KUKA KRL program: MyProgram_151().src

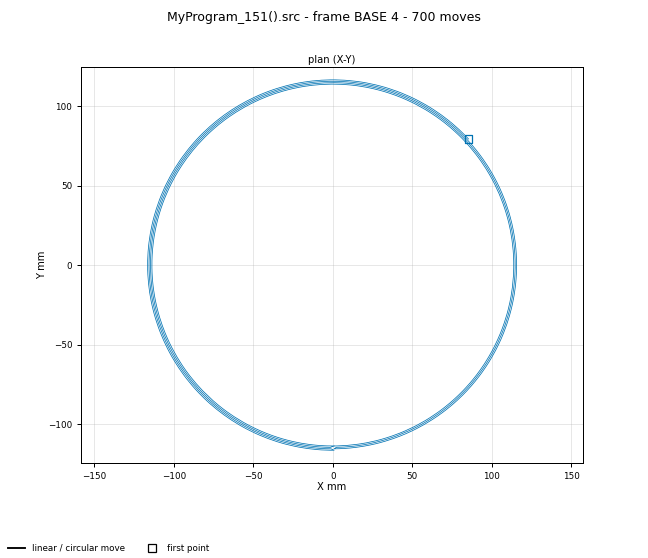
[picture p0: tool path of MyProgram_151().src in frame BASE 4, 700 of 700 moves have a stored position in this frame; points joined in program order, loops and branches not executed]
&ACCESS RVP
&REL 1
&PARAM TEMPLATE = C:\KRC\Roboter\Template\vorgabe
&PARAM EDITMASK = *
DEF MyProgram_151()
; ---- Setting reference (Base) ----
$BASE = BASE_DATA[4]

; --------------------------
; ---- Setting tool (TCP) ----
$TOOL = TOOL_DATA[3]
; --------------------------

$VEL.CP = VEL_APROX_PRINT
Startdeposition()
$VEL.CP = VEL_PRINT
LIN {X 85.3348,Y 79.272,Z 118,A 39.0033,B 24.9377,C -1.8229,E1 25.1164,E2 406.8947} C_DIS
LIN {X 83.3637,Y 81.3423,Z 118,A 40.3329,B 24.9377,C -1.8225,E1 25.1138,E2 405.572} C_DIS
LIN {X 81.214,Y 83.4873,Z 118,A 41.7921,B 24.9377,C -1.8241,E1 25.1109,E2 404.1151} C_DIS
LIN {X 79.272,Y 85.3348,Z 118,A 43.1327,B 24.9374,C -1.8278,E1 25.1082,E2 402.7712} C_DIS
LIN {X 76.7632,Y 87.5957,Z 118,A 44.7729,B 24.9372,C -1.8302,E1 25.1048,E2 401.1319} C_DIS
LIN {X 74.8522,Y 89.2356,Z 118,A 46.0205,B 24.937,C -1.833,E1 25.1021,E2 399.8825} C_DIS
LIN {X 72.6397,Y 91.0457,Z 118,A 47.421,B 24.9369,C -1.8354,E1 25.0991,E2 398.4816} C_DIS
LIN {X 70.3835,Y 92.8009,Z 118,A 48.9052,B 24.9364,C -1.8416,E1 25.0957,E2 396.9883} C_DIS
LIN {X 68.2299,Y 94.3968,Z 118,A 50.1353,B 24.9366,C -1.8398,E1 25.093,E2 395.7667} C_DIS
LIN {X 65.5697,Y 96.2615,Z 118,A 51.6474,B 24.9366,C -1.8386,E1 25.0895,E2 394.2626} C_DIS
LIN {X 63.3659,Y 97.7272,Z 118,A 53.0869,B 24.9361,C -1.847,E1 25.0861,E2 392.808} C_DIS
LIN {X 61.1008,Y 99.1603,Z 118,A 54.4098,B 24.9359,C -1.8492,E1 25.083,E2 391.4841} C_DIS
LIN {X 58.4944,Y 100.7187,Z 118,A 55.8287,B 24.9359,C -1.848,E1 25.0796,E2 390.0724} C_DIS
LIN {X 56.005,Y 102.1239,Z 118,A 57.3305,B 24.9355,C -1.8543,E1 25.0759,E2 388.56} C_DIS
LIN {X 53.6405,Y 103.3865,Z 118,A 58.5455,B 24.9358,C -1.8513,E1 25.0729,E2 387.3555} C_DIS
LIN {X 51.0872,Y 104.6717,Z 118,A 59.9607,B 24.9356,C -1.8535,E1 25.0694,E2 385.9389} C_DIS
LIN {X 48.503,Y 105.894,Z 118,A 61.3507,B 24.9356,C -1.8545,E1 25.0659,E2 384.5502} C_DIS
LIN {X 45.6034,Y 107.173,Z 118,A 62.7679,B 24.9359,C -1.8498,E1 25.0623,E2 383.1475} C_DIS
LIN {X 43.2486,Y 108.1463,Z 118,A 64.227,B 24.9351,C -1.8604,E1 25.0584,E2 381.6667} C_DIS
LIN {X 40.5815,Y 109.1751,Z 118,A 65.5599,B 24.9353,C -1.8584,E1 25.055,E2 380.3412} C_DIS
LIN {X 37.7211,Y 110.1951,Z 118,A 67.0508,B 24.9352,C -1.8596,E1 25.0511,E2 378.8505} C_DIS
LIN {X 35.1757,Y 111.0349,Z 118,A 68.4376,B 24.9349,C -1.8638,E1 25.0473,E2 377.4565} C_DIS
LIN {X 32.4402,Y 111.8647,Z 118,A 69.7714,B 24.935,C -1.8615,E1 25.0438,E2 376.1303} C_DIS
LIN {X 29.6851,Y 112.6271,Z 118,A 71.1757,B 24.935,C -1.8624,E1 25.04,E2 374.7262} C_DIS
LIN {X 26.9121,Y 113.3217,Z 118,A 72.58,B 24.935,C -1.8631,E1 25.0362,E2 373.3222} C_DIS
LIN {X 23.9484,Y 113.9839,Z 118,A 73.9931,B 24.9351,C -1.8603,E1 25.0324,E2 371.9178} C_DIS
LIN {X 21.3193,Y 114.5057,Z 118,A 75.4604,B 24.9346,C -1.8674,E1 25.0283,E2 370.4352} C_DIS
LIN {X 18.5028,Y 114.9944,Z 118,A 76.795,B 24.9348,C -1.8647,E1 25.0246,E2 369.1083} C_DIS
LIN {X 15.6751,Y 115.4139,Z 118,A 78.2709,B 24.9346,C -1.8682,E1 25.0205,E2 367.6255} C_DIS
LIN {X 12.6607,Y 115.7824,Z 118,A 79.6939,B 24.9348,C -1.8653,E1 25.0166,E2 366.2103} C_DIS
LIN {X 9.9931,Y 116.044,Z 118,A 81.1695,B 24.9343,C -1.8724,E1 25.0125,E2 364.7188} C_DIS
LIN {X 7.1422,Y 116.2543,Z 118,A 82.4182,B 24.9348,C -1.8654,E1 25.009,E2 363.4871} C_DIS
LIN {X 4.1089,Y 116.4,Z 118,A 83.9124,B 24.9348,C -1.8654,E1 25.0049,E2 361.9935} C_DIS
LIN {X 1.4293,Y 116.4647,Z 118,A 85.302,B 24.9346,C -1.8683,E1 25.001,E2 360.5972} C_DIS
LIN {X -1.4293,Y 116.4647,Z 118,A 86.6382,B 24.9348,C -1.8649,E1 24.9973,E2 359.2689} C_DIS
LIN {X -4.4651,Y 116.3869,Z 118,A 88.1333,B 24.9348,C -1.8645,E1 24.9931,E2 357.7745} C_DIS
LIN {X -7.1422,Y 116.2543,Z 118,A 89.5233,B 24.9346,C -1.8672,E1 24.9892,E2 356.378} C_DIS
LIN {X -10.1706,Y 116.0276,Z 118,A 90.9807,B 24.9348,C -1.8649,E1 24.9852,E2 354.9252} C_DIS
LIN {X -12.838,Y 115.7638,Z 118,A 92.3389,B 24.9348,C -1.8659,E1 24.9814,E2 353.5638} C_DIS
LIN {X -15.6751,Y 115.4139,Z 118,A 93.6765,B 24.935,C -1.862,E1 24.9777,E2 352.2345} C_DIS
LIN {X -18.5028,Y 114.9944,Z 118,A 95.0845,B 24.935,C -1.8611,E1 24.9738,E2 350.8273} C_DIS
LIN {X -21.3193,Y 114.5057,Z 118,A 96.4933,B 24.9351,C -1.8602,E1 24.9699,E2 349.4193} C_DIS
LIN {X -24.2971,Y 113.9101,Z 118,A 97.9106,B 24.9355,C -1.8556,E1 24.9661,E2 348.0112} C_DIS
LIN {X -27.0853,Y 113.2795,Z 118,A 99.3197,B 24.9355,C -1.8544,E1 24.9623,E2 346.6031} C_DIS
LIN {X -29.8571,Y 112.5806,Z 118,A 100.7287,B 24.9356,C -1.8532,E1 24.9585,E2 345.195} C_DIS
LIN {X -32.6721,Y 111.7959,Z 118,A 102.2246,B 24.9356,C -1.8541,E1 24.9544,E2 343.6945} C_DIS
LIN {X -35.3452,Y 110.98,Z 118,A 103.6275,B 24.9356,C -1.8537,E1 24.9507,E2 342.2901} C_DIS
LIN {X -38.0582,Y 110.0792,Z 118,A 105.0374,B 24.9356,C -1.8522,E1 24.947,E2 340.8812} C_DIS
LIN {X -40.7482,Y 109.112,Z 118,A 106.4477,B 24.9358,C -1.8505,E1 24.9433,E2 339.472} C_DIS
LIN {X -43.4137,Y 108.0791,Z 118,A 107.858,B 24.9359,C -1.8487,E1 24.9396,E2 338.0628} C_DIS
LIN {X -46.053,Y 106.9812,Z 118,A 109.2688,B 24.9361,C -1.8469,E1 24.936,E2 336.6532} C_DIS
LIN {X -48.6646,Y 105.8188,Z 118,A 110.6668,B 24.9362,C -1.8444,E1 24.9324,E2 335.2577} C_DIS
LIN {X -51.56,Y 104.4374,Z 118,A 112.0273,B 24.937,C -1.8327,E1 24.9291,E2 333.9215} C_DIS
LIN {X -53.8634,Y 103.2691,Z 118,A 113.5098,B 24.9366,C -1.8395,E1 24.9253,E2 332.4188} C_DIS
LIN {X -56.3172,Y 101.952,Z 118,A 114.9134,B 24.9366,C -1.8386,E1 24.9219,E2 331.0134} C_DIS
LIN {X -58.8023,Y 100.5392,Z 118,A 116.2454,B 24.937,C -1.8329,E1 24.9187,E2 329.6909} C_DIS
LIN {X -61.3804,Y 98.9856,Z 118,A 117.6643,B 24.9374,C -1.8276,E1 24.9153,E2 328.2803} C_DIS
LIN {X -63.5159,Y 97.631,Z 118,A 119.1322,B 24.9369,C -1.8346,E1 24.9118,E2 326.7911} C_DIS
LIN {X -66.0391,Y 95.9411,Z 118,A 120.5614,B 24.9373,C -1.8289,E1 24.9085,E2 325.3705} C_DIS
LIN {X -68.2299,Y 94.3968,Z 118,A 121.9567,B 24.9373,C -1.8294,E1 24.9054,E2 323.9693} C_DIS
LIN {X -70.6671,Y 92.5851,Z 118,A 123.3066,B 24.9379,C -1.8202,E1 24.9024,E2 322.6363} C_DIS
LIN {X -72.7796,Y 90.9352,Z 118,A 124.7114,B 24.9379,C -1.821,E1 24.8993,E2 321.2246} C_DIS
LIN {X -75.125,Y 89.0061,Z 118,A 126.2124,B 24.9381,C -1.8179,E1 24.8961,E2 319.7251} C_DIS
LIN {X -77.1539,Y 87.2545,Z 118,A 127.5376,B 24.9382,C -1.8152,E1 24.8933,E2 318.4011} C_DIS
LIN {X -79.5348,Y 85.0876,Z 118,A 128.9678,B 24.9389,C -1.8051,E1 24.8904,E2 316.9892} C_DIS
LIN {X -81.3423,Y 83.3637,Z 118,A 130.3644,B 24.9387,C -1.8091,E1 24.8875,E2 315.5773} C_DIS
LIN {X -83.3637,Y 81.3423,Z 118,A 131.8491,B 24.9387,C -1.8089,E1 24.8846,E2 314.0867} C_DIS
LIN {X -85.4553,Y 79.1407,Z 118,A 133.28,B 24.9391,C -1.8026,E1 24.8819,E2 312.6646} C_DIS
LIN {X -87.3718,Y 77.0196,Z 118,A 134.6941,B 24.9393,C -1.7993,E1 24.8793,E2 311.252} C_DIS
LIN {X -89.2356,Y 74.8522,Z 118,A 136.0285,B 24.9398,C -1.7927,E1 24.8769,E2 309.9273} C_DIS
LIN {X -90.9352,Y 72.7796,Z 118,A 137.4345,B 24.9398,C -1.7927,E1 24.8744,E2 308.5145} C_DIS
LIN {X -92.8009,Y 70.3835,Z 118,A 138.9372,B 24.94,C -1.7891,E1 24.8719,E2 307.0133} C_DIS
LIN {X -94.3968,Y 68.2299,Z 118,A 140.3345,B 24.94,C -1.7887,E1 24.8695,E2 305.6102} C_DIS
LIN {X -96.0428,Y 65.8928,Z 118,A 141.6783,B 24.9405,C -1.7822,E1 24.8674,E2 304.2753} C_DIS
LIN {X -97.7235,Y 63.3718,Z 118,A 143.1007,B 24.9409,C -1.7752,E1 24.8652,E2 302.8623} C_DIS
LIN {X -99.1603,Y 61.1008,Z 118,A 144.5079,B 24.9409,C -1.7749,E1 24.8632,E2 301.4487} C_DIS
LIN {X -100.7187,Y 58.4943,Z 118,A 146.0113,B 24.9412,C -1.771,E1 24.861,E2 299.9469} C_DIS
LIN {X -102.1239,Y 56.005,Z 118,A 147.4264,B 24.9415,C -1.7673,E1 24.8591,E2 298.5333} C_DIS
LIN {X -103.5905,Y 53.2413,Z 118,A 148.8412,B 24.9421,C -1.7576,E1 24.8573,E2 297.134} C_DIS
LIN {X -104.7489,Y 50.9265,Z 118,A 150.1771,B 24.9421,C -1.7563,E1 24.8556,E2 295.7939} C_DIS
LIN {X -105.894,Y 48.503,Z 118,A 151.5844,B 24.9422,C -1.7559,E1 24.854,E2 294.3799} C_DIS
LIN {X -107.1216,Y 45.7254,Z 118,A 153.0082,B 24.9427,C -1.7485,E1 24.8524,E2 292.966} C_DIS
LIN {X -108.1463,Y 43.2486,Z 118,A 154.4865,B 24.9425,C -1.751,E1 24.8508,E2 291.4735} C_DIS
LIN {X -109.1751,Y 40.5815,Z 118,A 155.8314,B 24.943,C -1.7441,E1 24.8495,E2 290.1375} C_DIS
LIN {X -110.1951,Y 37.7211,Z 118,A 157.335,B 24.9433,C -1.7398,E1 24.8481,E2 288.6355} C_DIS
LIN {X -111.0349,Y 35.1757,Z 118,A 158.7337,B 24.9433,C -1.7389,E1 24.8469,E2 287.2309} C_DIS
LIN {X -112.2544,Y 31.065,Z 118,A 160.8577,B 24.9437,C -1.7328,E1 24.8453,E2 285.1092} C_DIS
LIN {X -112.9829,Y 28.3007,Z 118,A 162.2735,B 24.944,C -1.7287,E1 24.8443,E2 283.695} C_DIS
LIN {X -113.6814,Y 25.3454,Z 118,A 163.7071,B 24.9445,C -1.7214,E1 24.8434,E2 282.2702} C_DIS
LIN {X -114.341,Y 22.175,Z 118,A 165.0605,B 24.9454,C -1.7065,E1 24.8427,E2 280.9443} C_DIS
LIN {X -114.7881,Y 19.7367,Z 118,A 166.4593,B 24.9452,C -1.7099,E1 24.842,E2 279.5293} C_DIS
LIN {X -115.2655,Y 16.7194,Z 118,A 168.0902,B 24.9452,C -1.7103,E1 24.8413,E2 277.8878} C_DIS
LIN {X -115.6183,Y 14.0806,Z 118,A 169.3713,B 24.9455,C -1.7048,E1 24.8408,E2 276.612} C_DIS
LIN {X -115.929,Y 11.2389,Z 118,A 170.7075,B 24.946,C -1.6974,E1 24.8405,E2 275.2856} C_DIS
LIN {X -116.1699,Y 8.3905,Z 118,A 172.1239,B 24.9463,C -1.6932,E1 24.8401,E2 273.8705} C_DIS
LIN {X -116.3408,Y 5.537,Z 118,A 173.6198,B 24.9463,C -1.6923,E1 24.8399,E2 272.3678} C_DIS
LIN {X -116.4384,Y 2.8584,Z 118,A 175.0528,B 24.9463,C -1.6927,E1 24.8399,E2 270.9254} C_DIS
LIN {X -116.4727,Y 0,Z 118,A 176.3346,B 24.9469,C -1.683,E1 24.8398,E2 269.6588} C_DIS
LIN {X -116.4384,Y -2.8584,Z 118,A 177.8509,B 24.9469,C -1.683,E1 24.8398,E2 268.1336} C_DIS
LIN {X -116.3233,Y -5.893,Z 118,A 179.2044,B 24.9476,C -1.6724,E1 24.84,E2 266.7971} C_DIS
LIN {X -116.1437,Y -8.746,Z 118,A -179.3796,B 24.9478,C -1.6682,E1 24.8403,E2 265.3825} C_DIS
LIN {X -115.9126,Y -11.4164,Z 118,A -177.9721,B 24.9478,C -1.6676,E1 24.8407,E2 263.968} C_DIS
LIN {X -115.5747,Y -14.4343,Z 118,A -176.5474,B 24.9484,C -1.66,E1 24.8411,E2 262.5529} C_DIS
LIN {X -115.2128,Y -17.0902,Z 118,A -175.14,B 24.9484,C -1.6594,E1 24.8417,E2 261.1385} C_DIS
LIN {X -114.7272,Y -20.0879,Z 118,A -173.6359,B 24.9487,C -1.6551,E1 24.8424,E2 259.6357} C_DIS
LIN {X -114.2355,Y -22.7228,Z 118,A -172.2374,B 24.9487,C -1.6543,E1 24.8431,E2 258.231} C_DIS
LIN {X -113.6434,Y -25.5195,Z 118,A -170.8217,B 24.949,C -1.6502,E1 24.844,E2 256.8166} C_DIS
LIN {X -112.9829,Y -28.3007,Z 118,A -169.406,B 24.9492,C -1.6463,E1 24.8449,E2 255.402} C_DIS
LIN {X -112.2544,Y -31.065,Z 118,A -168.0613,B 24.9496,C -1.6394,E1 24.8459,E2 254.066} C_DIS
LIN {X -111.4054,Y -33.9807,Z 118,A -166.5575,B 24.9499,C -1.6353,E1 24.8471,E2 252.5633} C_DIS
LIN {X -110.5379,Y -36.7045,Z 118,A -165.142,B 24.9501,C -1.6314,E1 24.8483,E2 251.149} C_DIS
LIN {X -109.6649,Y -39.2387,Z 118,A -163.7439,B 24.9501,C -1.6307,E1 24.8496,E2 249.7445} C_DIS
LIN {X -108.6038,Y -42.0841,Z 118,A -162.2321,B 24.9504,C -1.627,E1 24.8511,E2 248.2329} C_DIS
LIN {X -107.5068,Y -44.8114,Z 118,A -160.8878,B 24.9509,C -1.6186,E1 24.8525,E2 246.9012} C_DIS
LIN {X -106.408,Y -47.3623,Z 118,A -159.4815,B 24.951,C -1.6163,E1 24.8541,E2 245.4927} C_DIS
LIN {X -105.2908,Y -49.7988,Z 118,A -158.1547,B 24.9513,C -1.6129,E1 24.8557,E2 244.1668} C_DIS
LIN {X -104.0369,Y -52.3678,Z 118,A -156.6688,B 24.9513,C -1.6122,E1 24.8575,E2 242.6745} C_DIS
LIN {X -102.6355,Y -55.0619,Z 118,A -155.2369,B 24.9517,C -1.6055,E1 24.8594,E2 241.251} C_DIS
LIN {X -101.2533,Y -57.5641,Z 118,A -153.8226,B 24.9519,C -1.602,E1 24.8613,E2 239.8376} C_DIS
LIN {X -99.7679,Y -60.101,Z 118,A -152.3994,B 24.9522,C -1.5972,E1 24.8634,E2 238.4186} C_DIS
LIN {X -98.0992,Y -62.7864,Z 118,A -151.0558,B 24.953,C -1.5843,E1 24.8653,E2 237.0989} C_DIS
LIN {X -96.8442,Y -64.7092,Z 118,A -149.6679,B 24.9525,C -1.5921,E1 24.8675,E2 235.6854} C_DIS
LIN {X -94.9429,Y -67.4645,Z 118,A -148.2308,B 24.9533,C -1.5792,E1 24.8697,E2 234.272} C_DIS
LIN {X -93.5524,Y -69.3832,Z 118,A -146.7692,B 24.9527,C -1.5886,E1 24.8722,E2 232.7808} C_DIS
LIN {X -91.711,Y -71.798,Z 118,A -145.4181,B 24.9533,C -1.579,E1 24.8745,E2 231.4462} C_DIS
LIN {X -89.839,Y -74.1261,Z 118,A -143.9109,B 24.9533,C -1.5771,E1 24.8771,E2 229.9366} C_DIS
LIN {X -88.1947,Y -76.0773,Z 118,A -142.5998,B 24.9534,C -1.5765,E1 24.8795,E2 228.6209} C_DIS
LIN {X -86.3012,Y -78.2188,Z 118,A -141.0101,B 24.9532,C -1.5811,E1 24.8825,E2 227.0132} C_DIS
LIN {X -83.8978,Y -80.7881,Z 118,A -139.4276,B 24.9538,C -1.571,E1 24.8855,E2 225.4478} C_DIS
LIN {X -81.214,Y -83.4873,Z 118,A -137.5664,B 24.954,C -1.5665,E1 24.8892,E2 223.5894} C_DIS
LIN {X -79.1407,Y -85.4553,Z 118,A -136.0502,B 24.954,C -1.5683,E1 24.8923,E2 222.0628} C_DIS
LIN {X -77.0196,Y -87.3718,Z 118,A -134.8213,B 24.9545,C -1.5579,E1 24.8949,E2 220.8536} C_DIS
LIN {X -74.8522,Y -89.2356,Z 118,A -133.3295,B 24.9545,C -1.5589,E1 24.898,E2 219.3538} C_DIS
LIN {X -72.7796,Y -90.9352,Z 118,A -131.8718,B 24.9543,C -1.5623,E1 24.9012,E2 217.8824} C_DIS
LIN {X -70.3835,Y -92.8009,Z 118,A -130.5058,B 24.9547,C -1.5542,E1 24.9042,E2 216.5309} C_DIS
LIN {X -68.2299,Y -94.3968,Z 118,A -129.1117,B 24.9547,C -1.5551,E1 24.9074,E2 215.1296} C_DIS
LIN {X -65.7452,Y -96.1427,Z 118,A -127.6294,B 24.9549,C -1.5521,E1 24.9108,E2 213.6494} C_DIS
LIN {X -63.5159,Y -97.631,Z 118,A -126.36,B 24.9551,C -1.5479,E1 24.9137,E2 212.3859} C_DIS
LIN {X -60.7621,Y -99.3661,Z 118,A -124.9306,B 24.9557,C -1.5381,E1 24.9171,E2 210.9753} C_DIS
LIN {X -58.6489,Y -100.6299,Z 118,A -123.3921,B 24.955,C -1.5504,E1 24.9209,E2 209.4029} C_DIS
LIN {X -56.1616,Y -102.0389,Z 118,A -122.1279,B 24.9554,C -1.5423,E1 24.9239,E2 208.1543} C_DIS
LIN {X -53.4819,Y -103.4676,Z 118,A -120.63,B 24.9555,C -1.5406,E1 24.9276,E2 206.6564} C_DIS
LIN {X -50.9265,Y -104.7489,Z 118,A -119.2994,B 24.9558,C -1.5355,E1 24.9309,E2 205.3343} C_DIS
LIN {X -48.503,Y -105.894,Z 118,A -117.8549,B 24.9556,C -1.5395,E1 24.9346,E2 203.8768} C_DIS
LIN {X -45.8896,Y -107.0524,Z 118,A -116.4886,B 24.9558,C -1.5362,E1 24.9381,E2 202.5151} C_DIS
LIN {X -42.8981,Y -108.284,Z 118,A -115.0615,B 24.9563,C -1.5274,E1 24.9418,E2 201.1056} C_DIS
LIN {X -40.4141,Y -109.2362,Z 118,A -113.6618,B 24.9561,C -1.5302,E1 24.9454,E2 199.6965} C_DIS
LIN {X -37.89,Y -110.1382,Z 118,A -112.2614,B 24.956,C -1.5326,E1 24.9491,E2 198.2875} C_DIS
LIN {X -35.1757,Y -111.0349,Z 118,A -110.7822,B 24.9559,C -1.5347,E1 24.9531,E2 196.8007} C_DIS
LIN {X -32.2687,Y -111.9133,Z 118,A -109.4358,B 24.9563,C -1.5272,E1 24.9567,E2 195.4699} C_DIS
LIN {X -29.5125,Y -112.6715,Z 118,A -108.0277,B 24.9563,C -1.5264,E1 24.9605,E2 194.0615} C_DIS
LIN {X -26.5253,Y -113.4111,Z 118,A -106.6095,B 24.9566,C -1.5214,E1 24.9643,E2 192.6533} C_DIS
LIN {X -23.9484,Y -113.9839,Z 118,A -105.0271,B 24.956,C -1.5333,E1 24.9687,E2 191.0406} C_DIS
LIN {X -21.3193,Y -114.5057,Z 118,A -103.7426,B 24.956,C -1.5313,E1 24.9722,E2 189.7596} C_DIS
LIN {X -18.3266,Y -115.0217,Z 118,A -102.3183,B 24.9563,C -1.5277,E1 24.9761,E2 188.3423} C_DIS
LIN {X -15.6751,Y -115.4139,Z 118,A -100.9287,B 24.9561,C -1.5306,E1 24.98,E2 186.9448} C_DIS
LIN {X -12.6607,Y -115.7824,Z 118,A -99.5046,B 24.9563,C -1.5273,E1 24.9839,E2 185.5277} C_DIS
LIN {X -9.9931,Y -116.044,Z 118,A -98.1155,B 24.9561,C -1.5303,E1 24.9878,E2 184.1307} C_DIS
LIN {X -7.1422,Y -116.2543,Z 118,A -96.7798,B 24.9563,C -1.5272,E1 24.9915,E2 182.8019} C_DIS
LIN {X -4.1089,Y -116.4,Z 118,A -95.2861,B 24.9563,C -1.5274,E1 24.9957,E2 181.3075} C_DIS
LIN {X -1.4293,Y -116.4647,Z 118,A -93.8976,B 24.9561,C -1.5307,E1 24.9996,E2 179.9109} C_DIS
LIN {X 0.8178,Y -116.4663,Z 118,A -93.0487,B 24.9567,C -1.5195,E1 25.0019,E2 179.0887} C_DIS
Enddeposition()
LIN {X 0.8178,Y -116.4663,Z 118,A -93.0487,B 24.9567,C -1.5195,E1 25.0019,E2 179.0887} C_DIS
Startdeposition()
$VEL.CP = VEL_PRINT
LIN {X -1.1028,Y -115.5699,Z 118,A -94.4525,B 24.957,C -1.5148,E1 24.9979,E2 180.5035} C_DIS
LIN {X -4.4527,Y -115.4898,Z 118,A -96.1961,B 24.9572,C -1.511,E1 24.993,E2 182.2565} C_DIS
LIN {X -7.5005,Y -115.3312,Z 118,A -97.4691,B 24.9566,C -1.5215,E1 24.9895,E2 183.505} C_DIS
LIN {X -10.5343,Y -115.0934,Z 118,A -99.2856,B 24.9574,C -1.508,E1 24.9844,E2 185.3542} C_DIS
LIN {X -13.8894,Y -114.7377,Z 118,A -101.0033,B 24.9574,C -1.5063,E1 24.9796,E2 187.0772} C_DIS
LIN {X -17.3122,Y -114.271,Z 118,A -102.6849,B 24.9574,C -1.5081,E1 24.975,E2 188.756} C_DIS
LIN {X -20.8268,Y -113.6831,Z 118,A -104.3708,B 24.9572,C -1.5121,E1 24.9703,E2 190.4338} C_DIS
LIN {X -23.6853,Y -113.1224,Z 118,A -106.1192,B 24.9579,C -1.4996,E1 24.9655,E2 192.2141} C_DIS
LIN {X -30.1752,Y -111.5658,Z 118,A -109.089,B 24.9569,C -1.5161,E1 24.9575,E2 195.1489} C_DIS
LIN {X -33.1484,Y -110.7191,Z 118,A -110.6752,B 24.957,C -1.5148,E1 24.9533,E2 196.7407} C_DIS
LIN {X -36.3666,Y -109.7054,Z 118,A -112.2338,B 24.9567,C -1.521,E1 24.9491,E2 198.2875} C_DIS
LIN {X -39.5147,Y -108.6096,Z 118,A -113.9421,B 24.9567,C -1.5201,E1 24.9446,E2 200.0013} C_DIS
LIN {X -42.6548,Y -107.4161,Z 118,A -115.6122,B 24.9567,C -1.5215,E1 24.9403,E2 201.6717} C_DIS
LIN {X -45.0198,Y -106.4457,Z 118,A -117.2427,B 24.9574,C -1.5073,E1 24.936,E2 203.3394} C_DIS
LIN {X -49.5351,Y -104.4225,Z 118,A -119.4741,B 24.9567,C -1.5195,E1 24.9304,E2 205.5474} C_DIS
LIN {X -55.2689,Y -101.5029,Z 118,A -122.5886,B 24.9563,C -1.5269,E1 24.9227,E2 208.653} C_DIS
LIN {X -58.6758,Y -99.5723,Z 118,A -124.6398,B 24.9564,C -1.525,E1 24.9177,E2 210.7147} C_DIS
LIN {X -61.3742,Y -97.9321,Z 118,A -126.1678,B 24.9562,C -1.529,E1 24.9141,E2 212.2382} C_DIS
LIN {X -64.8345,Y -95.6763,Z 118,A -128.2313,B 24.9561,C -1.5316,E1 24.9093,E2 214.3021} C_DIS
LIN {X -67.7046,Y -93.6699,Z 118,A -129.8549,B 24.9556,C -1.5392,E1 24.9056,E2 215.9133} C_DIS
LIN {X -69.8641,Y -92.0694,Z 118,A -131.1535,B 24.9554,C -1.543,E1 24.9027,E2 217.2075} C_DIS
LIN {X -72.7677,Y -89.7905,Z 118,A -133.1001,B 24.9554,C -1.5415,E1 24.8984,E2 219.1648} C_DIS
LIN {X -75.7652,Y -87.2767,Z 118,A -135.072,B 24.9554,C -1.5439,E1 24.8943,E2 221.1387} C_DIS
LIN {X -78.7575,Y -84.5874,Z 118,A -137.8065,B 24.9569,C -1.5175,E1 24.8885,E2 223.9471} C_DIS
LIN {X -82.3524,Y -81.0899,Z 118,A -139.5208,B 24.9547,C -1.5546,E1 24.8853,E2 225.5805} C_DIS
LIN {X -84.8214,Y -78.505,Z 118,A -141.3998,B 24.9547,C -1.5541,E1 24.8817,E2 227.4689} C_DIS
LIN {X -87.4411,Y -75.5769,Z 118,A -143.2564,B 24.9543,C -1.5623,E1 24.8783,E2 229.3144} C_DIS
LIN {X -89.0171,Y -73.712,Z 118,A -144.5314,B 24.9543,C -1.5625,E1 24.876,E2 230.5947} C_DIS
LIN {X -93.7328,Y -67.6164,Z 118,A -148.2256,B 24.9534,C -1.577,E1 24.8698,E2 234.272} C_DIS
LIN {X -96.5065,Y -63.5921,Z 118,A -150.8312,B 24.9534,C -1.5758,E1 24.8656,E2 236.8934} C_DIS
LIN {X -99.1104,Y -59.4561,Z 118,A -153.1405,B 24.9528,C -1.5868,E1 24.8622,E2 239.1883} C_DIS
LIN {X -100.4168,Y -57.2197,Z 118,A -154.436,B 24.9526,C -1.5898,E1 24.8604,E2 240.4834} C_DIS
LIN {X -102.1313,Y -54.0992,Z 118,A -156.3555,B 24.9527,C -1.5884,E1 24.8579,E2 242.4163} C_DIS
LIN {X -103.5428,Y -51.3455,Z 118,A -157.8376,B 24.9523,C -1.5948,E1 24.856,E2 243.8911} C_DIS
LIN {X -104.9905,Y -48.3187,Z 118,A -159.6176,B 24.9523,C -1.5948,E1 24.8539,E2 245.6808} C_DIS
LIN {X -106.851,Y -44.0521,Z 118,A -161.8498,B 24.9518,C -1.6046,E1 24.8515,E2 247.9021} C_DIS
LIN {X -109.2746,Y -37.6424,Z 118,A -165.3336,B 24.9514,C -1.6111,E1 24.8481,E2 251.3899} C_DIS
LIN {X -110.5899,Y -33.5827,Z 118,A -167.302,B 24.9506,C -1.6235,E1 24.8465,E2 253.3402} C_DIS
LIN {X -111.2894,Y -31.1809,Z 118,A -168.5648,B 24.9504,C -1.6264,E1 24.8455,E2 254.6033} C_DIS
LIN {X -112.2235,Y -27.6296,Z 118,A -170.5441,B 24.9504,C -1.6257,E1 24.8441,E2 256.5959} C_DIS
LIN {X -113.1797,Y -23.4059,Z 118,A -172.6582,B 24.95,C -1.6337,E1 24.8429,E2 258.7034} C_DIS
LIN {X -113.8153,Y -20.0916,Z 118,A -174.2534,B 24.9495,C -1.6421,E1 24.8421,E2 260.288} C_DIS
LIN {X -114.6692,Y -14.4427,Z 118,A -177.486,B 24.9499,C -1.6351,E1 24.8408,E2 263.5564} C_DIS
LIN {X -115.0302,Y -11.2176,Z 118,A -178.9568,B 24.9492,C -1.6458,E1 24.8404,E2 265.0107} C_DIS
LIN {X -115.2891,Y -8.1231,Z 118,A 178.9077,B 24.9504,C -1.6272,E1 24.84,E2 267.2035} C_DIS
LIN {X -115.538,Y -2.9602,Z 118,A 177.1917,B 24.9478,C -1.669,E1 24.8398,E2 268.83} C_DIS
LIN {X -115.5741,Y -0.3375,Z 118,A 175.4733,B 24.9486,C -1.6566,E1 24.8398,E2 270.5884} C_DIS
LIN {X -115.54,Y 2.8967,Z 118,A 173.4408,B 24.9493,C -1.6448,E1 24.84,E2 272.6611} C_DIS
LIN {X -115.3136,Y 7.761,Z 118,A 172.1171,B 24.9461,C -1.696,E1 24.8402,E2 273.8707} C_DIS
LIN {X -114.6731,Y 14.4126,Z 118,A 168.5235,B 24.9461,C -1.6955,E1 24.8412,E2 277.4871} C_DIS
LIN {X -114.1151,Y 18.3208,Z 118,A 166.2604,B 24.9465,C -1.6896,E1 24.8421,E2 279.7776} C_DIS
LIN {X -113.3576,Y 22.5391,Z 118,A 164.157,B 24.946,C -1.6973,E1 24.8432,E2 281.8752} C_DIS
LIN {X -112.5714,Y 26.1758,Z 118,A 162.3427,B 24.9456,C -1.7045,E1 24.8443,E2 283.683} C_DIS
LIN {X -111.7231,Y 29.5927,Z 118,A 160.5855,B 24.9452,C -1.7096,E1 24.8455,E2 285.4384} C_DIS
LIN {X -110.7368,Y 33.0887,Z 118,A 158.7588,B 24.9449,C -1.7143,E1 24.847,E2 287.2644} C_DIS
LIN {X -109.6222,Y 36.6133,Z 118,A 156.624,B 24.9453,C -1.7081,E1 24.8488,E2 289.4263} C_DIS
LIN {X -108.4715,Y 39.8935,Z 118,A 155.328,B 24.9439,C -1.7304,E1 24.85,E2 290.6762} C_DIS
LIN {X -107.3461,Y 42.8328,Z 118,A 153.7534,B 24.9436,C -1.7347,E1 24.8516,E2 292.2495} C_DIS
LIN {X -105.1499,Y 47.9712,Z 118,A 151.1031,B 24.9427,C -1.748,E1 24.8546,E2 294.8829} C_DIS
LIN {X -103.1967,Y 52.0412,Z 118,A 148.5805,B 24.943,C -1.7433,E1 24.8577,E2 297.4302} C_DIS
LIN {X -101.5405,Y 55.1997,Z 118,A 146.8619,B 24.9426,C -1.7505,E1 24.8599,E2 299.1407} C_DIS
LIN {X -99.9869,Y 57.9679,Z 118,A 145.3976,B 24.942,C -1.7595,E1 24.8619,E2 300.5912} C_DIS
LIN {X -97.3396,Y 62.3095,Z 118,A 143.0997,B 24.9409,C -1.7757,E1 24.8653,E2 302.8623} C_DIS
LIN {X -95.1302,Y 65.6343,Z 118,A 140.6772,B 24.9417,C -1.7634,E1 24.8691,E2 305.3262} C_DIS
LIN {X -91.8464,Y 70.1565,Z 118,A 137.9139,B 24.9412,C -1.7713,E1 24.8737,E2 308.0841} C_DIS
LIN {X -89.4004,Y 73.2489,Z 118,A 136.1221,B 24.9404,C -1.783,E1 24.8768,E2 309.8563} C_DIS
LIN {X -87.4387,Y 75.5797,Z 118,A 134.6337,B 24.9401,C -1.7878,E1 24.8794,E2 311.34} C_DIS
LIN {X -85.255,Y 78.0324,Z 118,A 132.8543,B 24.9402,C -1.7859,E1 24.8828,E2 313.132} C_DIS
LIN {X -83.1023,Y 80.3211,Z 118,A 131.2447,B 24.9402,C -1.7876,E1 24.8859,E2 314.7443} C_DIS
LIN {X -80.8004,Y 82.6384,Z 118,A 129.5894,B 24.9399,C -1.7901,E1 24.8892,E2 316.4008} C_DIS
LIN {X -78.2147,Y 85.0878,Z 118,A 127.8643,B 24.9395,C -1.7959,E1 24.8927,E2 318.119} C_DIS
LIN {X -75.8248,Y 87.2246,Z 118,A 126.396,B 24.939,C -1.8045,E1 24.8957,E2 319.5727} C_DIS
LIN {X -73.823,Y 88.9248,Z 118,A 124.9212,B 24.9392,C -1.8004,E1 24.8989,E2 321.063} C_DIS
LIN {X -71.2386,Y 91.01,Z 118,A 123.2058,B 24.9392,C -1.8011,E1 24.9027,E2 322.783} C_DIS
LIN {X -67.7823,Y 93.613,Z 118,A 121.2713,B 24.9383,C -1.8142,E1 24.907,E2 324.6932} C_DIS
LIN {X -65.909,Y 94.9393,Z 118,A 120.1272,B 24.9382,C -1.8163,E1 24.9096,E2 325.8363} C_DIS
LIN {X -63.1122,Y 96.8229,Z 118,A 118.3935,B 24.9382,C -1.817,E1 24.9136,E2 327.5741} C_DIS
LIN {X -60.2848,Y 98.6068,Z 118,A 116.7068,B 24.938,C -1.8189,E1 24.9177,E2 329.2614} C_DIS
LIN {X -57.2261,Y 100.4131,Z 118,A 114.9657,B 24.9377,C -1.8229,E1 24.9218,E2 330.9983} C_DIS
LIN {X -52.3371,Y 103.0455,Z 118,A 112.2026,B 24.9374,C -1.8271,E1 24.9287,E2 333.759} C_DIS
LIN {X -47.7074,Y 105.2688,Z 118,A 109.7972,B 24.9367,C -1.837,E1 24.9347,E2 336.1471} C_DIS
LIN {X -45.0225,Y 106.4446,Z 118,A 108.1349,B 24.9372,C -1.8304,E1 24.939,E2 337.829} C_DIS
LIN {X -39.8705,Y 108.4799,Z 118,A 105.3791,B 24.937,C -1.8337,E1 24.9462,E2 340.5828} C_DIS
LIN {X -36.146,Y 109.7783,Z 118,A 103.5675,B 24.9364,C -1.8421,E1 24.9509,E2 342.3779} C_DIS
LIN {X -33.9409,Y 110.4788,Z 118,A 102.2176,B 24.9369,C -1.8349,E1 24.9546,E2 343.7471} C_DIS
LIN {X -30.0619,Y 111.5964,Z 118,A 100.3173,B 24.9364,C -1.8413,E1 24.9596,E2 345.6353} C_DIS
LIN {X -26.5782,Y 112.4784,Z 118,A 98.3889,B 24.9368,C -1.8368,E1 24.9649,E2 347.577} C_DIS
LIN {X -20.5619,Y 113.7307,Z 118,A 95.421,B 24.9364,C -1.8427,E1 24.973,E2 350.5344} C_DIS
LIN {X -16.5537,Y 114.3832,Z 118,A 92.8961,B 24.9377,C -1.8224,E1 24.9801,E2 353.1094} C_DIS
LIN {X -12.4409,Y 114.9037,Z 118,A 91.5096,B 24.9357,C -1.8519,E1 24.9838,E2 354.4269} C_DIS
LIN {X -9.586,Y 115.1769,Z 118,A 89.6331,B 24.937,C -1.8332,E1 24.9891,E2 356.3486} C_DIS
LIN {X -5.0728,Y 115.4631,Z 118,A 87.7327,B 24.9359,C -1.8486,E1 24.9943,E2 358.2131} C_DIS
LIN {X -1.7778,Y 115.5613,Z 118,A 86.1165,B 24.9359,C -1.8498,E1 24.9988,E2 359.8265} C_DIS
LIN {X 2.7921,Y 115.5416,Z 118,A 83.7219,B 24.9362,C -1.8446,E1 25.0055,E2 362.2332} C_DIS
LIN {X 5.6487,Y 115.4384,Z 118,A 82.3078,B 24.9362,C -1.8448,E1 25.0095,E2 363.6464} C_DIS
LIN {X 9.3531,Y 115.1955,Z 118,A 80.5288,B 24.936,C -1.8474,E1 25.0144,E2 365.4184} C_DIS
LIN {X 12.566,Y 114.8906,Z 118,A 78.9724,B 24.936,C -1.849,E1 25.0187,E2 366.9699} C_DIS
LIN {X 16.9867,Y 114.3214,Z 118,A 76.7453,B 24.936,C -1.8477,E1 25.0249,E2 369.1982} C_DIS
LIN {X 20.4012,Y 113.7596,Z 118,A 74.9773,B 24.9362,C -1.8449,E1 25.0298,E2 370.9711} C_DIS
LIN {X 23.1806,Y 113.226,Z 118,A 73.0282,B 24.9379,C -1.8205,E1 25.0353,E2 372.9756} C_DIS
LIN {X 27.4736,Y 112.2616,Z 118,A 71.4536,B 24.9361,C -1.8457,E1 25.0394,E2 374.4883} C_DIS
LIN {X 31.3419,Y 111.2438,Z 118,A 69.4296,B 24.9364,C -1.8426,E1 25.0448,E2 376.5164} C_DIS
LIN {X 34.7917,Y 110.215,Z 118,A 67.5714,B 24.9367,C -1.8379,E1 25.0498,E2 378.3822} C_DIS
LIN {X 38.1071,Y 109.1116,Z 118,A 65.9663,B 24.9364,C -1.8421,E1 25.054,E2 379.9744} C_DIS
LIN {X 41.1391,Y 108.005,Z 118,A 64.4543,B 24.9362,C -1.8444,E1 25.058,E2 381.4776} C_DIS
LIN {X 44.3693,Y 106.7199,Z 118,A 62.7798,B 24.9362,C -1.8448,E1 25.0623,E2 383.1475} C_DIS
LIN {X 46.695,Y 105.723,Z 118,A 61.4611,B 24.9365,C -1.8405,E1 25.0657,E2 384.473} C_DIS
LIN {X 49.414,Y 104.4806,Z 118,A 59.4893,B 24.9381,C -1.817,E1 25.0708,E2 386.4954} C_DIS
LIN {X 52.535,Y 102.9443,Z 118,A 58.5493,B 24.9359,C -1.8498,E1 25.0729,E2 387.3554} C_DIS
LIN {X 54.9269,Y 101.6884,Z 118,A 56.9024,B 24.9369,C -1.8342,E1 25.0771,E2 389.0346} C_DIS
LIN {X 57.7827,Y 100.0933,Z 118,A 55.1828,B 24.9374,C -1.8275,E1 25.0813,E2 390.7648} C_DIS
LIN {X 60.6472,Y 98.3862,Z 118,A 53.4633,B 24.9378,C -1.8219,E1 25.0854,E2 392.4921} C_DIS
LIN {X 64.2244,Y 96.089,Z 118,A 51.5795,B 24.9373,C -1.8286,E1 25.0897,E2 394.3539} C_DIS
LIN {X 67.7372,Y 93.646,Z 118,A 49.2623,B 24.9382,C -1.8161,E1 25.0951,E2 396.6925} C_DIS
LIN {X 70.6895,Y 91.4357,Z 118,A 47.4842,B 24.9382,C -1.8151,E1 25.099,E2 398.4666} C_DIS
LIN {X 74.3331,Y 88.501,Z 118,A 45.3378,B 24.938,C -1.8185,E1 25.1036,E2 400.5968} C_DIS
LIN {X 76.5967,Y 86.5496,Z 118,A 43.3045,B 24.9399,C -1.7906,E1 25.108,E2 402.688} C_DIS
LIN {X 79.3369,Y 84.0426,Z 118,A 41.9401,B 24.9387,C -1.8084,E1 25.1107,E2 404.0048} C_DIS
LIN {X 82.398,Y 81.0438,Z 118,A 39.9218,B 24.9387,C -1.8086,E1 25.1147,E2 406.0139} C_DIS
LIN {X 84.7171,Y 78.6177,Z 118,A 37.93,B 24.9399,C -1.7899,E1 25.1186,E2 408.0412} C_DIS
LIN {X 87.8428,Y 75.1075,Z 118,A 35.8955,B 24.9394,C -1.7981,E1 25.1222,E2 410.0474} C_DIS
LIN {X 89.8531,Y 72.6903,Z 118,A 33.9847,B 24.9407,C -1.7782,E1 25.1257,E2 411.9961} C_DIS
LIN {X 92.5392,Y 69.2388,Z 118,A 32.1823,B 24.94,C -1.7896,E1 25.1287,E2 413.7631} C_DIS
LIN {X 94.2757,Y 66.8555,Z 118,A 30.7553,B 24.9401,C -1.7876,E1 25.131,E2 415.188} C_DIS
LIN {X 97.0918,Y 62.6957,Z 118,A 28.4569,B 24.9399,C -1.79,E1 25.1346,E2 417.4693} C_DIS
LIN {X 98.3355,Y 60.7284,Z 118,A 26.9266,B 24.9413,C -1.7695,E1 25.1369,E2 419.0403} C_DIS
LIN {X 100.4042,Y 57.2417,Z 118,A 25.0707,B 24.9413,C -1.7712,E1 25.1395,E2 420.8827} C_DIS
LIN {X 101.7139,Y 54.8799,Z 118,A 23.7124,B 24.9415,C -1.7666,E1 25.1413,E2 422.2447} C_DIS
LIN {X 103.2359,Y 51.9646,Z 118,A 21.9385,B 24.9423,C -1.7553,E1 25.1435,E2 424.0357} C_DIS
LIN {X 105.0661,Y 48.1554,Z 118,A 19.9713,B 24.9423,C -1.7553,E1 25.1459,E2 425.9924} C_DIS
LIN {X 106.4671,Y 44.9692,Z 118,A 18.2492,B 24.9426,C -1.7504,E1 25.1478,E2 427.7165} C_DIS
LIN {X 108.0684,Y 40.9717,Z 118,A 16.194,B 24.9427,C -1.7478,E1 25.1499,E2 429.7664} C_DIS
LIN {X 109.1301,Y 38.0542,Z 118,A 14.7568,B 24.9427,C -1.748,E1 25.1512,E2 431.1952} C_DIS
LIN {X 110.1706,Y 34.9337,Z 118,A 13.1212,B 24.9431,C -1.7428,E1 25.1526,E2 432.8338} C_DIS
LIN {X 110.8806,Y 32.6042,Z 118,A 11.9037,B 24.9433,C -1.7386,E1 25.1536,E2 434.0541} C_DIS
LIN {X 111.6032,Y 30.0365,Z 118,A 10.5501,B 24.9437,C -1.7331,E1 25.1546,E2 435.4131} C_DIS
LIN {X 112.6196,Y 25.9668,Z 118,A 7.9783,B 24.9456,C -1.7036,E1 25.1563,E2 438.0394} C_DIS
LIN {X 113.4391,Y 22.1157,Z 118,A 6.4426,B 24.9448,C -1.7169,E1 25.1571,E2 439.5348} C_DIS
LIN {X 114.2092,Y 17.7119,Z 118,A 4.2818,B 24.945,C -1.7124,E1 25.1581,E2 441.6935} C_DIS
LIN {X 114.7865,Y 13.4726,Z 118,A 2.1673,B 24.9455,C -1.706,E1 25.1588,E2 443.8107} C_DIS
LIN {X 115.1106,Y 10.3478,Z 118,A 0.7122,B 24.9455,C -1.7057,E1 25.1592,E2 445.2578} C_DIS
LIN {X 115.3397,Y 7.3753,Z 118,A -0.8389,B 24.946,C -1.6975,E1 25.1595,E2 446.819} C_DIS
LIN {X 115.5005,Y 4.1836,Z 118,A -2.2668,B 24.9459,C -1.6997,E1 25.1597,E2 448.2333} C_DIS
LIN {X 115.5578,Y 1.9702,Z 118,A -3.4879,B 24.9465,C -1.6904,E1 25.1597,E2 449.4691} C_DIS
LIN {X 115.5656,Y -1.5443,Z 118,A -5.1785,B 24.9467,C -1.6871,E1 25.1597,E2 451.1574} C_DIS
LIN {X 115.5005,Y -4.1753,Z 118,A -6.3896,B 24.9467,C -1.6872,E1 25.1597,E2 452.3609} C_DIS
LIN {X 115.2855,Y -8.177,Z 118,A -8.3536,B 24.947,C -1.6818,E1 25.1593,E2 454.326} C_DIS
LIN {X 115.0258,Y -11.2666,Z 118,A -10.079,B 24.9479,C -1.6679,E1 25.1589,E2 456.074} C_DIS
LIN {X 114.7122,Y -14.1072,Z 118,A -11.5025,B 24.9482,C -1.663,E1 25.1584,E2 457.5007} C_DIS
LIN {X 114.1154,Y -18.319,Z 118,A -13.4016,B 24.948,C -1.666,E1 25.1576,E2 459.3815} C_DIS
LIN {X 113.6328,Y -21.1062,Z 118,A -14.9504,B 24.9487,C -1.6545,E1 25.1569,E2 460.9483} C_DIS
LIN {X 112.9006,Y -24.7167,Z 118,A -16.7041,B 24.9489,C -1.6521,E1 25.1558,E2 462.6975} C_DIS
LIN {X 112.1708,Y -27.8459,Z 118,A -18.4645,B 24.9497,C -1.6391,E1 25.1547,E2 464.4784} C_DIS
LIN {X 111.0734,Y -31.9432,Z 118,A -20.398,B 24.9496,C -1.6403,E1 25.1532,E2 466.398} C_DIS
LIN {X 110.2542,Y -34.6652,Z 118,A -21.6954,B 24.9496,C -1.6411,E1 25.1522,E2 467.6861} C_DIS
LIN {X 109.4265,Y -37.1938,Z 118,A -22.963,B 24.9496,C -1.6393,E1 25.1511,E2 468.9507} C_DIS
LIN {X 108.2948,Y -40.3738,Z 118,A -24.6168,B 24.9499,C -1.635,E1 25.1495,E2 470.6054} C_DIS
LIN {X 107.3498,Y -42.8236,Z 118,A -26.1676,B 24.9509,C -1.6192,E1 25.1479,E2 472.1849} C_DIS
LIN {X 105.8897,Y -46.3126,Z 118,A -27.8831,B 24.9508,C -1.6209,E1 25.146,E2 473.8869} C_DIS
LIN {X 104.3166,Y -49.7556,Z 118,A -30.3361,B 24.9527,C -1.5883,E1 25.143,E2 476.4036} C_DIS
LIN {X 102.3793,Y -53.6283,Z 118,A -32.6142,B 24.9535,C -1.5758,E1 25.14,E2 478.6992} C_DIS
LIN {X 99.9494,Y -58.0332,Z 118,A -34.7455,B 24.9529,C -1.5853,E1 25.1371,E2 480.7971} C_DIS
LIN {X 98.2034,Y -60.9399,Z 118,A -36.1544,B 24.9524,C -1.5931,E1 25.1351,E2 482.1804} C_DIS
LIN {X 96.1407,Y -64.1468,Z 118,A -38.0411,B 24.9528,C -1.5879,E1 25.1322,E2 484.0701} C_DIS
LIN {X 93.6333,Y -67.7546,Z 118,A -39.9821,B 24.9525,C -1.5929,E1 25.1291,E2 485.9898} C_DIS
LIN {X 92.1435,Y -69.7655,Z 118,A -41.4132,B 24.9532,C -1.5806,E1 25.1266,E2 487.443} C_DIS
LIN {X 89.52,Y -73.1014,Z 118,A -43.3724,B 24.9532,C -1.5817,E1 25.1232,E2 489.3904} C_DIS
LIN {X 87.007,Y -76.074,Z 118,A -45.4033,B 24.9537,C -1.5719,E1 25.1195,E2 491.4351} C_DIS
LIN {X 84.2424,Y -79.1245,Z 118,A -47.3206,B 24.9537,C -1.5725,E1 25.1159,E2 493.3427} C_DIS
LIN {X 81.6698,Y -81.7796,Z 118,A -49.0726,B 24.9537,C -1.5716,E1 25.1125,E2 495.0892} C_DIS
LIN {X 79.7374,Y -83.6649,Z 118,A -50.4352,B 24.954,C -1.5673,E1 25.1098,E2 496.4565} C_DIS
LIN {X 78.0971,Y -85.1956,Z 118,A -51.5624,B 24.9542,C -1.564,E1 25.1074,E2 497.5869} C_DIS
LIN {X 76.0421,Y -87.0348,Z 118,A -52.8745,B 24.9542,C -1.5633,E1 25.1047,E2 498.8953} C_DIS
LIN {X 73.7975,Y -88.946,Z 118,A -54.4733,B 24.9548,C -1.5536,E1 25.1013,E2 500.5107} C_DIS
LIN {X 71.1341,Y -91.0925,Z 118,A -56.0457,B 24.9547,C -1.5556,E1 25.0978,E2 502.0727} C_DIS
LIN {X 69.0629,Y -92.6713,Z 118,A -57.5088,B 24.9553,C -1.5449,E1 25.0945,E2 503.5558} C_DIS
LIN {X 66.0239,Y -94.8594,Z 118,A -59.2953,B 24.9553,C -1.5443,E1 25.0905,E2 505.3375} C_DIS
LIN {X 62.4463,Y -97.2519,Z 118,A -61.4262,B 24.9556,C -1.5402,E1 25.0855,E2 507.4711} C_DIS
LIN {X 59.6223,Y -99.0094,Z 118,A -62.9137,B 24.9553,C -1.5444,E1 25.082,E2 508.9439} C_DIS
LIN {X 57.5032,Y -100.2539,Z 118,A -64.3045,B 24.9559,C -1.5343,E1 25.0786,E2 510.3543} C_DIS
LIN {X 54.5546,Y -101.8903,Z 118,A -65.8252,B 24.9557,C -1.5383,E1 25.0749,E2 511.8613} C_DIS
LIN {X 52.5489,Y -102.9372,Z 118,A -67.1906,B 24.9564,C -1.5253,E1 25.0714,E2 513.2536} C_DIS
LIN {X 49.7556,Y -104.3166,Z 118,A -68.6477,B 24.9564,C -1.5267,E1 25.0678,E2 514.7036} C_DIS
LIN {X 45.9403,Y -106.052,Z 118,A -71.1927,B 24.9577,C -1.5025,E1 25.0611,E2 517.2997} C_DIS
LIN {X 41.9944,Y -107.6755,Z 118,A -72.8241,B 24.9566,C -1.5213,E1 25.057,E2 518.883} C_DIS
LIN {X 37.9621,Y -109.1624,Z 118,A -74.8032,B 24.9564,C -1.5253,E1 25.0519,E2 520.8485} C_DIS
LIN {X 35.3644,Y -110.0312,Z 118,A -76.1021,B 24.9564,C -1.5263,E1 25.0484,E2 522.1426} C_DIS
LIN {X 32.939,Y -110.7813,Z 118,A -77.5484,B 24.9569,C -1.5164,E1 25.0445,E2 523.6098} C_DIS
LIN {X 29.4365,Y -111.765,Z 118,A -79.1855,B 24.9566,C -1.5219,E1 25.0401,E2 525.2313} C_DIS
LIN {X 26.8101,Y -112.4235,Z 118,A -80.9741,B 24.9578,C -1.5006,E1 25.0351,E2 527.0677} C_DIS
LIN {X 23.5929,Y -113.1413,Z 118,A -82.0109,B 24.9564,C -1.5258,E1 25.0325,E2 528.0434} C_DIS
LIN {X 19.6063,Y -113.9003,Z 118,A -84.5701,B 24.9579,C -1.4997,E1 25.0253,E2 530.6616} C_DIS
LIN {X 14.838,Y -114.618,Z 118,A -86.6646,B 24.9572,C -1.5112,E1 25.0196,E2 532.7269} C_DIS
LIN {X 10.8564,Y -115.0637,Z 118,A -88.7021,B 24.9574,C -1.5078,E1 25.0139,E2 534.7711} C_DIS
LIN {X 7.7448,Y -115.3147,Z 118,A -90.1863,B 24.9573,C -1.5099,E1 25.0098,E2 536.2497} C_DIS
LIN {X 3.9505,Y -115.5076,Z 118,A -91.8465,B 24.9568,C -1.5191,E1 25.0052,E2 537.8877} C_DIS
LIN {X 0.8166,Y -115.5716,Z 118,A -92.8133,B 24.9553,C -1.5447,E1 25.0027,E2 538.7935} C_DIS
Enddeposition()
LIN {X 0.8166,Y -115.5716,Z 118,A -92.8133,B 24.9553,C -1.5447,E1 25.0027,E2 538.7935} C_DIS
Startdeposition()
$VEL.CP = VEL_PRINT
LIN {X 2.2158,Y -114.6563,Z 118,A -92.2661,B 24.9548,C -1.5537,E1 25.0043,E2 538.225} C_DIS
LIN {X 7.1921,Y -114.4532,Z 118,A -89.645,B 24.9544,C -1.5606,E1 25.0116,E2 535.5886} C_DIS
LIN {X 13.0705,Y -113.9307,Z 118,A -86.7386,B 24.9544,C -1.5603,E1 25.0197,E2 532.6847} C_DIS
LIN {X 16.1316,Y -113.5374,Z 118,A -85.2018,B 24.9544,C -1.5611,E1 25.0239,E2 531.1473} C_DIS
LIN {X 19.5457,Y -113.0015,Z 118,A -83.469,B 24.9542,C -1.5626,E1 25.0287,E2 529.4125} C_DIS
LIN {X 22.2221,Y -112.5048,Z 118,A -81.5172,B 24.9526,C -1.5906,E1 25.0343,E2 527.397} C_DIS
LIN {X 26.4977,Y -111.5766,Z 118,A -79.8033,B 24.9537,C -1.5712,E1 25.0388,E2 525.7313} C_DIS
LIN {X 30.5946,Y -110.5231,Z 118,A -77.7029,B 24.9537,C -1.5729,E1 25.0444,E2 523.6303} C_DIS
LIN {X 33.4389,Y -109.6955,Z 118,A -76.2531,B 24.9537,C -1.5732,E1 25.0483,E2 522.1822} C_DIS
LIN {X 37.1888,Y -108.4818,Z 118,A -74.4786,B 24.954,C -1.5669,E1 25.053,E2 520.4262} C_DIS
LIN {X 40.7064,Y -107.2099,Z 118,A -72.5661,B 24.9537,C -1.5714,E1 25.058,E2 518.507} C_DIS
LIN {X 48.0612,Y -104.1211,Z 118,A -68.5484,B 24.9533,C -1.5787,E1 25.0683,E2 514.4816} C_DIS
LIN {X 52.8911,Y -101.7535,Z 118,A -65.8332,B 24.953,C -1.5844,E1 25.0751,E2 511.7603} C_DIS
LIN {X 55.3245,Y -100.452,Z 118,A -64.4081,B 24.9527,C -1.5889,E1 25.0786,E2 510.3286} C_DIS
LIN {X 58.3616,Y -98.7162,Z 118,A -62.7326,B 24.9527,C -1.5889,E1 25.0827,E2 508.6583} C_DIS
LIN {X 61.3762,Y -96.8726,Z 118,A -60.9561,B 24.9525,C -1.5927,E1 25.0869,E2 506.8783} C_DIS
LIN {X 66.1386,Y -93.6855,Z 118,A -58.1252,B 24.9522,C -1.597,E1 25.0934,E2 504.0469} C_DIS
LIN {X 68.7427,Y -91.7901,Z 118,A -56.5701,B 24.9522,C -1.5979,E1 25.0969,E2 502.4952} C_DIS
LIN {X 71.5425,Y -89.6267,Z 118,A -54.7033,B 24.9516,C -1.6064,E1 25.101,E2 500.6153} C_DIS
LIN {X 74.299,Y -87.3534,Z 118,A -53.0225,B 24.9516,C -1.6056,E1 25.1046,E2 498.9428} C_DIS
LIN {X 76.8055,Y -85.159,Z 118,A -51.2456,B 24.9511,C -1.6147,E1 25.1083,E2 497.1516} C_DIS
LIN {X 79.463,Y -82.6839,Z 118,A -49.5064,B 24.9511,C -1.6156,E1 25.1119,E2 495.4174} C_DIS
LIN {X 82.2743,Y -79.8879,Z 118,A -47.5434,B 24.9508,C -1.6197,E1 25.1157,E2 493.4532} C_DIS
LIN {X 84.5628,Y -77.4604,Z 118,A -45.8667,B 24.9506,C -1.6244,E1 25.1189,E2 491.7728} C_DIS
LIN {X 87.2007,Y -74.4783,Z 118,A -43.9466,B 24.9504,C -1.6263,E1 25.1224,E2 489.8567} C_DIS
LIN {X 89.3835,Y -71.8454,Z 118,A -42.1573,B 24.9499,C -1.6346,E1 25.1256,E2 488.0561} C_DIS
LIN {X 92.5207,Y -67.7561,Z 118,A -39.6714,B 24.9498,C -1.6375,E1 25.1298,E2 485.5752} C_DIS
LIN {X 94.5716,Y -64.8663,Z 118,A -37.8841,B 24.9494,C -1.6432,E1 25.1326,E2 483.7832} C_DIS
LIN {X 96.2831,Y -62.2952,Z 118,A -35.9796,B 24.9481,C -1.6647,E1 25.1356,E2 481.8376} C_DIS
LIN {X 98.0984,Y -59.3944,Z 118,A -34.7047,B 24.949,C -1.6491,E1 25.1374,E2 480.6059} C_DIS
LIN {X 100.1786,Y -55.8141,Z 118,A -32.4963,B 24.9483,C -1.6618,E1 25.1404,E2 478.3791} C_DIS
LIN {X 102.0212,Y -52.3706,Z 118,A -30.6715,B 24.9483,C -1.6617,E1 25.1428,E2 476.5643} C_DIS
LIN {X 103.8813,Y -48.5766,Z 118,A -28.582,B 24.9479,C -1.667,E1 25.1453,E2 474.4733} C_DIS
LIN {X 105.9782,Y -43.8175,Z 118,A -25.9035,B 24.9472,C -1.6788,E1 25.1483,E2 471.7818} C_DIS
LIN {X 107.2711,Y -40.5448,Z 118,A -24.2444,B 24.9472,C -1.6796,E1 25.15,E2 470.1299} C_DIS
LIN {X 108.5555,Y -36.97,Z 118,A -22.344,B 24.9467,C -1.6857,E1 25.1517,E2 468.2259} C_DIS
LIN {X 110.1935,Y -31.7589,Z 118,A -19.6387,B 24.9463,C -1.6932,E1 25.1539,E2 465.5182} C_DIS
LIN {X 110.9867,Y -28.8621,Z 118,A -18.0087,B 24.9456,C -1.7042,E1 25.1551,E2 463.8718} C_DIS
LIN {X 112.2146,Y -23.6476,Z 118,A -15.408,B 24.9453,C -1.7092,E1 25.1567,E2 461.2744} C_DIS
LIN {X 112.9973,Y -19.5708,Z 118,A -12.86,B 24.9434,C -1.7385,E1 25.158,E2 458.6723} C_DIS
LIN {X 113.6521,Y -15.313,Z 118,A -11.2777,B 24.9447,C -1.7183,E1 25.1585,E2 457.1467} C_DIS
LIN {X 114.2561,Y -9.8482,Z 118,A -8.4922,B 24.944,C -1.7291,E1 25.1593,E2 454.3524} C_DIS
LIN {X 114.5112,Y -6.1786,Z 118,A -6.8457,B 24.9442,C -1.7261,E1 25.1596,E2 452.7228} C_DIS
LIN {X 114.6665,Y -1.6593,Z 118,A -4.2823,B 24.9427,C -1.7478,E1 25.1598,E2 450.1233} C_DIS
LIN {X 114.6334,Y 3.1996,Z 118,A -2.0789,B 24.9429,C -1.7451,E1 25.1597,E2 447.9395} C_DIS
LIN {X 114.5017,Y 6.3506,Z 118,A -0.3422,B 24.9421,C -1.7578,E1 25.1594,E2 446.1831} C_DIS
LIN {X 114.0487,Y 11.9943,Z 118,A 2.2025,B 24.9424,C -1.7535,E1 25.1588,E2 443.6637} C_DIS
LIN {X 113.7052,Y 14.9034,Z 118,A 3.7604,B 24.9418,C -1.7627,E1 25.1583,E2 442.0934} C_DIS
LIN {X 112.6219,Y 21.6167,Z 118,A 6.9622,B 24.9417,C -1.7642,E1 25.1568,E2 438.9068} C_DIS
LIN {X 111.4288,Y 27.1032,Z 118,A 9.8759,B 24.9407,C -1.778,E1 25.155,E2 435.9774} C_DIS
LIN {X 110.5155,Y 30.6223,Z 118,A 11.762,B 24.9402,C -1.7869,E1 25.1536,E2 434.0813} C_DIS
LIN {X 109.6542,Y 33.5722,Z 118,A 13.2639,B 24.9399,C -1.79,E1 25.1524,E2 432.5806} C_DIS
LIN {X 108.587,Y 36.8767,Z 118,A 15.0092,B 24.9396,C -1.7957,E1 25.1509,E2 430.8316} C_DIS
LIN {X 106.4751,Y 42.5962,Z 118,A 18.1035,B 24.9388,C -1.807,E1 25.1478,E2 427.728} C_DIS
LIN {X 105.0275,Y 46.0462,Z 118,A 19.7758,B 24.9391,C -1.8032,E1 25.146,E2 426.0737} C_DIS
LIN {X 102.4348,Y 51.5613,Z 118,A 22.9996,B 24.9379,C -1.8202,E1 25.142,E2 422.8272} C_DIS
LIN {X 100.7074,Y 54.8545,Z 118,A 24.6915,B 24.9381,C -1.8176,E1 25.1398,E2 421.1503} C_DIS
LIN {X 98.8537,Y 58.1289,Z 118,A 26.575,B 24.9377,C -1.8229,E1 25.1372,E2 419.2641} C_DIS
LIN {X 96.9399,Y 61.2697,Z 118,A 28.2848,B 24.9377,C -1.8218,E1 25.1347,E2 417.5654} C_DIS
LIN {X 95.1205,Y 64.0557,Z 118,A 30.1304,B 24.9369,C -1.8347,E1 25.1318,E2 415.6987} C_DIS
LIN {X 92.7328,Y 67.4663,Z 118,A 32.1225,B 24.9369,C -1.8358,E1 25.1286,E2 413.7135} C_DIS
LIN {X 90.8592,Y 69.9684,Z 118,A 34.8247,B 24.9328,C -1.8929,E1 25.1238,E2 410.8894} C_DIS
LIN {X 86.5229,Y 75.2649,Z 118,A 37.8174,B 24.9337,C -1.8808,E1 25.1184,E2 407.9388} C_DIS
LIN {X 83.1064,Y 79.0233,Z 118,A 39.6236,B 24.9357,C -1.8525,E1 25.1151,E2 406.2072} C_DIS
LIN {X 80.6413,Y 81.535,Z 118,A 41.3743,B 24.9354,C -1.856,E1 25.1116,E2 404.4557} C_DIS
LIN {X 75.1121,Y 86.6563,Z 118,A 45.1082,B 24.935,C -1.8622,E1 25.1039,E2 400.7223} C_DIS
LIN {X 71.431,Y 89.7148,Z 118,A 47.4754,B 24.9348,C -1.8656,E1 25.0988,E2 398.356} C_DIS
LIN {X 68.6904,Y 91.8295,Z 118,A 49.2283,B 24.9345,C -1.8698,E1 25.0949,E2 396.5995} C_DIS
LIN {X 66.1409,Y 93.6839,Z 118,A 50.8735,B 24.934,C -1.8757,E1 25.0911,E2 394.9461} C_DIS
LIN {X 62.7541,Y 95.9848,Z 118,A 52.7553,B 24.9343,C -1.8717,E1 25.0868,E2 393.0802} C_DIS
LIN {X 60.1937,Y 97.6121,Z 118,A 54.3443,B 24.9339,C -1.8773,E1 25.083,E2 391.4829} C_DIS
LIN {X 58.1583,Y 98.8363,Z 118,A 55.8526,B 24.9328,C -1.8936,E1 25.0793,E2 389.9406} C_DIS
LIN {X 55.2435,Y 100.4964,Z 118,A 57.2922,B 24.9334,C -1.8853,E1 25.0758,E2 388.525} C_DIS
LIN {X 51.4272,Y 102.5013,Z 118,A 60.3446,B 24.9303,C -1.9287,E1 25.068,E2 385.378} C_DIS
LIN {X 45.8306,Y 105.1215,Z 118,A 62.2468,B 24.9338,C -1.8788,E1 25.0634,E2 383.5986} C_DIS
LIN {X 41.4229,Y 106.9364,Z 118,A 64.9005,B 24.9328,C -1.8934,E1 25.0565,E2 380.9166} C_DIS
LIN {X 37.3646,Y 108.4217,Z 118,A 67.0703,B 24.9326,C -1.8958,E1 25.0508,E2 378.7454} C_DIS
LIN {X 33.4066,Y 109.7055,Z 118,A 69.1052,B 24.9326,C -1.8955,E1 25.0454,E2 376.715} C_DIS
LIN {X 30.0083,Y 110.6819,Z 118,A 70.7881,B 24.9328,C -1.893,E1 25.0409,E2 375.0407} C_DIS
LIN {X 26.4711,Y 111.5827,Z 118,A 72.7387,B 24.9324,C -1.8996,E1 25.0355,E2 373.0772} C_DIS
LIN {X 22.2553,Y 112.4989,Z 118,A 75.1976,B 24.9313,C -1.914,E1 25.0287,E2 370.5873} C_DIS
LIN {X 18.7112,Y 113.141,Z 118,A 76.6069,B 24.9325,C -1.8975,E1 25.025,E2 369.2186} C_DIS
LIN {X 12.6062,Y 113.9846,Z 118,A 79.6861,B 24.9325,C -1.8981,E1 25.0164,E2 366.1404} C_DIS
LIN {X 8.4778,Y 114.3658,Z 118,A 81.8204,B 24.9323,C -1.901,E1 25.0105,E2 364.0005} C_DIS
LIN {X 5.1833,Y 114.5607,Z 118,A 83.8873,B 24.931,C -1.9192,E1 25.0046,E2 361.8911} C_DIS
LIN {X 1.0735,Y 114.6732,Z 118,A 85.3386,B 24.9328,C -1.8927,E1 25.0007,E2 360.5028} C_DIS
LIN {X -5.3564,Y 114.5533,Z 118,A 88.2915,B 24.9337,C -1.8805,E1 24.9926,E2 357.5783} C_DIS
LIN {X -12.221,Y 114.0249,Z 118,A 91.5458,B 24.9344,C -1.871,E1 24.9836,E2 354.3454} C_DIS
LIN {X -18.581,Y 113.1628,Z 118,A 95.0378,B 24.9337,C -1.8809,E1 24.9738,E2 350.8271} C_DIS
LIN {X -20.575,Y 112.8171,Z 118,A 96.9139,B 24.9311,C -1.9171,E1 24.9684,E2 348.8632} C_DIS
LIN {X -25.0213,Y 111.9163,Z 118,A 98.6606,B 24.9328,C -1.8928,E1 24.9638,E2 347.172} C_DIS
LIN {X -28.9604,Y 110.9614,Z 118,A 100.6365,B 24.9331,C -1.8887,E1 24.9585,E2 345.2029} C_DIS
LIN {X -34.1097,Y 109.4875,Z 118,A 103.2273,B 24.9336,C -1.8822,E1 24.9516,E2 342.6234} C_DIS
LIN {X -37.6193,Y 108.3323,Z 118,A 105.1905,B 24.9334,C -1.8848,E1 24.9463,E2 340.6502} C_DIS
LIN {X -44.3587,Y 105.7511,Z 118,A 108.578,B 24.9344,C -1.8707,E1 24.9376,E2 337.2889} C_DIS
LIN {X -50.1804,Y 103.1175,Z 118,A 112.0015,B 24.9341,C -1.8754,E1 24.9289,E2 333.8459} C_DIS
LIN {X -52.9233,Y 101.737,Z 118,A 113.9657,B 24.933,C -1.8908,E1 24.9239,E2 331.8397} C_DIS
LIN {X -56.2617,Y 99.9287,Z 118,A 115.6572,B 24.9338,C -1.8789,E1 24.9198,E2 330.1716} C_DIS
LIN {X -60.4702,Y 97.4393,Z 118,A 117.7614,B 24.9351,C -1.8603,E1 24.9149,E2 328.1051} C_DIS
LIN {X -64.9949,Y 94.4824,Z 118,A 120.725,B 24.9347,C -1.8658,E1 24.908,E2 325.1186} C_DIS
LIN {X -68.3635,Y 92.075,Z 118,A 122.6386,B 24.9355,C -1.8551,E1 24.9037,E2 323.2237} C_DIS
LIN {X -71.4311,Y 89.7147,Z 118,A 124.516,B 24.9359,C -1.8486,E1 24.8996,E2 321.3549} C_DIS
LIN {X -74.6893,Y 87.021,Z 118,A 126.8817,B 24.9355,C -1.8543,E1 24.8945,E2 318.9665} C_DIS
LIN {X -77.7869,Y 84.2631,Z 118,A 128.8088,B 24.9363,C -1.8435,E1 24.8905,E2 317.0574} C_DIS
LIN {X -80.2585,Y 81.9131,Z 118,A 130.5912,B 24.9363,C -1.8426,E1 24.8869,E2 315.2696} C_DIS
LIN {X -83.7641,Y 78.324,Z 118,A 133.3926,B 24.936,C -1.8485,E1 24.8815,E2 312.4422} C_DIS
LIN {X -86.0663,Y 75.7877,Z 118,A 134.8402,B 24.937,C -1.8333,E1 24.8789,E2 311.0242} C_DIS
LIN {X -88.7656,Y 72.6078,Z 118,A 136.6986,B 24.938,C -1.8187,E1 24.8756,E2 309.1922} C_DIS
LIN {X -91.9844,Y 68.4842,Z 118,A 139.3883,B 24.9383,C -1.8147,E1 24.871,E2 306.4992} C_DIS
LIN {X -94.4573,Y 65.0296,Z 118,A 141.7929,B 24.9379,C -1.8202,E1 24.8671,E2 304.0695} C_DIS
LIN {X -96.758,Y 61.5554,Z 118,A 144.2044,B 24.9374,C -1.8277,E1 24.8634,E2 301.628} C_DIS
LIN {X -98.8155,Y 58.1936,Z 118,A 145.6322,B 24.9393,C -1.8,E1 24.8615,E2 300.2588} C_DIS
LIN {X -100.3568,Y 55.4951,Z 118,A 147.456,B 24.9388,C -1.8064,E1 24.8589,E2 298.4102} C_DIS
LIN {X -102.4375,Y 51.5559,Z 118,A 149.5061,B 24.9398,C -1.7927,E1 24.8564,E2 296.3819} C_DIS
LIN {X -104.1478,Y 48.0039,Z 118,A 152.6528,B 24.9369,C -1.8346,E1 24.8526,E2 293.1179} C_DIS
LIN {X -106.8715,Y 41.5881,Z 118,A 154.7851,B 24.9414,C -1.769,E1 24.8505,E2 291.1304} C_DIS
LIN {X -108.9061,Y 35.9283,Z 118,A 158.086,B 24.9412,C -1.7714,E1 24.8474,E2 287.805} C_DIS
LIN {X -109.9648,Y 32.5379,Z 118,A 159.7749,B 24.9418,C -1.7623,E1 24.846,E2 286.1279} C_DIS
LIN {X -111.0101,Y 28.7711,Z 118,A 161.708,B 24.9423,C -1.7553,E1 24.8446,E2 284.2003} C_DIS
LIN {X -111.8656,Y 25.2464,Z 118,A 163.6684,B 24.9423,C -1.7553,E1 24.8434,E2 282.2282} C_DIS
LIN {X -112.6076,Y 21.691,Z 118,A 165.3633,B 24.9429,C -1.7448,E1 24.8425,E2 280.5486} C_DIS
LIN {X -113.2501,Y 18.0457,Z 118,A 167.3834,B 24.9429,C -1.7456,E1 24.8415,E2 278.5145} C_DIS
LIN {X -113.7716,Y 14.391,Z 118,A 169.2017,B 24.9434,C -1.7386,E1 24.8409,E2 276.7021} C_DIS
LIN {X -114.2613,Y 9.7844,Z 118,A 171.5425,B 24.9438,C -1.7321,E1 24.8402,E2 274.3628} C_DIS
LIN {X -114.4782,Y 6.7748,Z 118,A 173.4488,B 24.943,C -1.7433,E1 24.8399,E2 272.4183} C_DIS
LIN {X -114.6438,Y 2.8627,Z 118,A 175.6861,B 24.9427,C -1.7483,E1 24.8398,E2 270.1555} C_DIS
LIN {X -114.6588,Y -2.0793,Z 118,A 177.3829,B 24.9453,C -1.709,E1 24.8398,E2 268.5422} C_DIS
LIN {X -114.3427,Y -8.7659,Z 118,A -178.5349,B 24.944,C -1.7281,E1 24.8406,E2 264.39} C_DIS
LIN {X -113.8909,Y -13.4105,Z 118,A -176.8838,B 24.9463,C -1.693,E1 24.841,E2 262.8126} C_DIS
LIN {X -113.4873,Y -16.4838,Z 118,A -175.1879,B 24.9463,C -1.694,E1 24.8417,E2 261.1043} C_DIS
LIN {X -112.8673,Y -20.2964,Z 118,A -173.3849,B 24.9469,C -1.6828,E1 24.8425,E2 259.3174} C_DIS
LIN {X -112.1313,Y -24.0354,Z 118,A -171.464,B 24.9473,C -1.6775,E1 24.8436,E2 257.3977} C_DIS
LIN {X -111.4341,Y -27.0815,Z 118,A -169.9126,B 24.9476,C -1.6722,E1 24.8446,E2 255.8498} C_DIS
LIN {X -110.5556,Y -30.4757,Z 118,A -168.0633,B 24.9476,C -1.6707,E1 24.846,E2 253.9932} C_DIS
LIN {X -109.5927,Y -33.7703,Z 118,A -166.1831,B 24.9476,C -1.6722,E1 24.8475,E2 252.0986} C_DIS
LIN {X -108.4111,Y -37.3949,Z 118,A -164.114,B 24.9476,C -1.6732,E1 24.8494,E2 250.0154} C_DIS
LIN {X -106.4233,Y -42.7241,Z 118,A -161.5859,B 24.9489,C -1.652,E1 24.8519,E2 247.5237} C_DIS
LIN {X -105.0424,Y -46.0118,Z 118,A -159.8421,B 24.9493,C -1.6453,E1 24.8538,E2 245.7862} C_DIS
LIN {X -103.6062,Y -49.1633,Z 118,A -157.961,B 24.9493,C -1.6465,E1 24.856,E2 243.892} C_DIS
LIN {X -102.1303,Y -52.1571,Z 118,A -155.8112,B 24.9483,C -1.6616,E1 24.8588,E2 241.6945} C_DIS
LIN {X -100.1114,Y -55.9345,Z 118,A -154.2522,B 24.9501,C -1.6319,E1 24.8608,E2 240.1983} C_DIS
LIN {X -98.2038,Y -59.221,Z 118,A -152.5441,B 24.9509,C -1.619,E1 24.8632,E2 238.5121} C_DIS
LIN {X -95.5729,Y -63.3789,Z 118,A -149.8002,B 24.9506,C -1.6242,E1 24.8674,E2 235.7417} C_DIS
LIN {X -93.0689,Y -67.0029,Z 118,A -147.3598,B 24.9503,C -1.6285,E1 24.8714,E2 233.2792} C_DIS
LIN {X -89.5462,Y -71.6444,Z 118,A -144.6207,B 24.9512,C -1.6143,E1 24.876,E2 230.5609} C_DIS
LIN {X -87.2542,Y -74.4155,Z 118,A -142.3964,B 24.9503,C -1.6279,E1 24.8801,E2 228.2941} C_DIS
LIN {X -84.6044,Y -77.415,Z 118,A -140.8762,B 24.9518,C -1.6034,E1 24.8829,E2 226.8255} C_DIS
LIN {X -82.2201,Y -79.9442,Z 118,A -138.9855,B 24.9517,C -1.606,E1 24.8866,E2 224.9205} C_DIS
LIN {X -77.0396,Y -84.9489,Z 118,A -135.4341,B 24.9522,C -1.5965,E1 24.8938,E2 221.377} C_DIS
LIN {X -74.2781,Y -87.3713,Z 118,A -133.6515,B 24.9526,C -1.5908,E1 24.8975,E2 219.6011} C_DIS
LIN {X -71.1165,Y -89.9634,Z 118,A -131.6121,B 24.9528,C -1.5868,E1 24.9019,E2 217.5635} C_DIS
LIN {X -67.1792,Y -92.9431,Z 118,A -128.9158,B 24.9525,C -1.5921,E1 24.908,E2 214.845} C_DIS
LIN {X -63.2455,Y -95.6608,Z 118,A -126.722,B 24.9532,C -1.58,E1 24.9131,E2 212.6727} C_DIS
LIN {X -57.8274,Y -99.0319,Z 118,A -123.4792,B 24.9534,C -1.5775,E1 24.9208,E2 209.4258} C_DIS
LIN {X -54.218,Y -101.0527,Z 118,A -120.733,B 24.9518,C -1.6039,E1 24.9278,E2 206.6092} C_DIS
LIN {X -49.7002,Y -103.3482,Z 118,A -118.8584,B 24.9537,C -1.5725,E1 24.9323,E2 204.8043} C_DIS
LIN {X -47.1966,Y -104.5153,Z 118,A -117.23,B 24.9531,C -1.5816,E1 24.9365,E2 203.1503} C_DIS
LIN {X -44.15,Y -105.8391,Z 118,A -115.8942,B 24.9541,C -1.5659,E1 24.9398,E2 201.8487} C_DIS
LIN {X -40.1329,Y -107.4271,Z 118,A -113.6586,B 24.954,C -1.5672,E1 24.9457,E2 199.6053} C_DIS
LIN {X -36.7385,Y -108.6336,Z 118,A -111.9603,B 24.9543,C -1.5613,E1 24.9501,E2 197.9178} C_DIS
LIN {X -33.1791,Y -109.7746,Z 118,A -110.0392,B 24.9543,C -1.5622,E1 24.9553,E2 195.9913} C_DIS
LIN {X -29.2854,Y -110.8772,Z 118,A -107.9122,B 24.9541,C -1.5655,E1 24.961,E2 193.8532} C_DIS
LIN {X -25.4506,Y -111.8184,Z 118,A -106.0226,B 24.9544,C -1.5608,E1 24.9661,E2 191.972} C_DIS
LIN {X -21.2372,Y -112.6949,Z 118,A -103.8969,B 24.9544,C -1.5589,E1 24.972,E2 189.8485} C_DIS
LIN {X -16.1099,Y -113.5405,Z 118,A -101.127,B 24.9541,C -1.5658,E1 24.9797,E2 187.0598} C_DIS
LIN {X -12.0534,Y -114.0425,Z 118,A -99.3282,B 24.9547,C -1.5548,E1 24.9846,E2 185.2859} C_DIS
LIN {X -9.2264,Y -114.3059,Z 118,A -97.9502,B 24.9548,C -1.5529,E1 24.9884,E2 183.9116} C_DIS
LIN {X -4.8934,Y -114.5732,Z 118,A -95.3571,B 24.9537,C -1.5718,E1 24.9958,E2 181.2731} C_DIS
LIN {X -1.5627,Y -114.6683,Z 118,A -93.9277,B 24.9543,C -1.5617,E1 24.9997,E2 179.8677} C_DIS
LIN {X -1.5627,Y -114.6683,Z 118,A -93.9277,B 24.9543,C -1.5617,E1 24.9997,E2 179.8677} C_DIS
Enddeposition()
LIN {X 0.8048,Y -113.7717,Z 118,A -93.5798,B 24.9555,C -1.5411,E1 25.0005,E2 179.5686} C_DIS
Startdeposition()
$VEL.CP = VEL_PRINT
LIN {X -3.7511,Y -113.7193,Z 118,A -96.5887,B 24.9573,C -1.5099,E1 24.9919,E2 182.6517} C_DIS
LIN {X -8.2771,Y -113.481,Z 118,A -98.3158,B 24.9559,C -1.5336,E1 24.9873,E2 184.3233} C_DIS
LIN {X -10.9246,Y -113.2561,Z 118,A -100.1097,B 24.957,C -1.5142,E1 24.9822,E2 186.1641} C_DIS
LIN {X -14.8946,Y -112.802,Z 118,A -102.3544,B 24.9576,C -1.5048,E1 24.9759,E2 188.4328} C_DIS
LIN {X -19.8773,Y -112.0314,Z 118,A -104.8743,B 24.9575,C -1.5065,E1 24.9689,E2 190.9513} C_DIS
LIN {X -24.7754,Y -111.052,Z 118,A -106.5714,B 24.9554,C -1.5422,E1 24.9645,E2 192.5658} C_DIS
LIN {X -28.698,Y -110.1029,Z 118,A -108.7715,B 24.9558,C -1.5362,E1 24.9585,E2 194.7832} C_DIS
LIN {X -32.0023,Y -109.1882,Z 118,A -110.4106,B 24.9555,C -1.541,E1 24.9541,E2 196.4134} C_DIS
LIN {X -35.0986,Y -108.232,Z 118,A -112.1004,B 24.9555,C -1.5399,E1 24.9496,E2 198.1091} C_DIS
LIN {X -38.6746,Y -107.0068,Z 118,A -113.7173,B 24.9548,C -1.5536,E1 24.9454,E2 199.6965} C_DIS
LIN {X -42.358,Y -105.604,Z 118,A -115.8192,B 24.955,C -1.5505,E1 24.9399,E2 201.8102} C_DIS
LIN {X -45.2656,Y -104.3894,Z 118,A -117.511,B 24.9551,C -1.5478,E1 24.9356,E2 203.5123} C_DIS
LIN {X -48.758,Y -102.806,Z 118,A -120.2224,B 24.9568,C -1.5177,E1 24.9285,E2 206.302} C_DIS
LIN {X -53.1593,Y -100.5991,Z 118,A -121.9297,B 24.9548,C -1.5528,E1 24.9245,E2 207.9306} C_DIS
LIN {X -56.2488,Y -98.9061,Z 118,A -123.5772,B 24.9544,C -1.5605,E1 24.9205,E2 209.5647} C_DIS
LIN {X -61.9505,Y -95.4387,Z 118,A -127.0366,B 24.9544,C -1.5614,E1 24.9122,E2 213.0326} C_DIS
LIN {X -66.6538,Y -92.2162,Z 118,A -130.1278,B 24.9546,C -1.5571,E1 24.9051,E2 216.1445} C_DIS
LIN {X -69.6023,Y -90.009,Z 118,A -131.83,B 24.954,C -1.5667,E1 24.9014,E2 217.8301} C_DIS
LIN {X -72.3848,Y -87.7878,Z 118,A -133.7164,B 24.954,C -1.5662,E1 24.8972,E2 219.7247} C_DIS
LIN {X -75.2502,Y -85.345,Z 118,A -135.6263,B 24.9539,C -1.5694,E1 24.8932,E2 221.6346} C_DIS
LIN {X -81.8571,Y -79.0285,Z 118,A -139.8315,B 24.9523,C -1.5952,E1 24.8849,E2 225.7958} C_DIS
LIN {X -85.983,Y -74.5197,Z 118,A -143.3753,B 24.953,C -1.5832,E1 24.8781,E2 229.3839} C_DIS
LIN {X -88.3813,Y -71.6577,Z 118,A -145.1334,B 24.9525,C -1.5926,E1 24.875,E2 231.1278} C_DIS
LIN {X -89.9342,Y -69.6995,Z 118,A -146.9834,B 24.9537,C -1.572,E1 24.8718,E2 233.0358} C_DIS
LIN {X -92.4049,Y -66.3894,Z 118,A -148.4776,B 24.952,C -1.6005,E1 24.8694,E2 234.4691} C_DIS
LIN {X -94.6291,Y -63.1811,Z 118,A -151.4839,B 24.9542,C -1.5643,E1 24.8646,E2 237.5767} C_DIS
LIN {X -97.7961,Y -58.1557,Z 118,A -153.2514,B 24.9508,C -1.6207,E1 24.8622,E2 239.2188} C_DIS
LIN {X -101.177,Y -52.0518,Z 118,A -157.047,B 24.9508,C -1.619,E1 24.8571,E2 243.0384} C_DIS
LIN {X -102.8586,Y -48.6485,Z 118,A -159.0396,B 24.9508,C -1.6212,E1 24.8546,E2 245.0367} C_DIS
LIN {X -104.0437,Y -46.0587,Z 118,A -160.5242,B 24.9506,C -1.6233,E1 24.853,E2 246.5244} C_DIS
LIN {X -105.5495,Y -42.492,Z 118,A -162.2333,B 24.9497,C -1.6386,E1 24.8512,E2 248.2067} C_DIS
LIN {X -107.1722,Y -38.2169,Z 118,A -164.68,B 24.9497,C -1.6397,E1 24.8488,E2 250.6646} C_DIS
LIN {X -108.9117,Y -32.9344,Z 118,A -167.5047,B 24.9492,C -1.6472,E1 24.8464,E2 253.4876} C_DIS
LIN {X -109.7617,Y -29.9756,Z 118,A -169.1573,B 24.9492,C -1.6479,E1 24.8451,E2 255.1479} C_DIS
LIN {X -110.7924,Y -25.9079,Z 118,A -171.2002,B 24.9485,C -1.6573,E1 24.8438,E2 257.1806} C_DIS
LIN {X -111.5179,Y -22.5817,Z 118,A -173.008,B 24.9485,C -1.659,E1 24.8427,E2 258.995} C_DIS
LIN {X -112.1225,Y -19.3645,Z 118,A -174.4659,B 24.9476,C -1.6716,E1 24.842,E2 260.4313} C_DIS
LIN {X -112.7284,Y -15.45,Z 118,A -176.6847,B 24.9478,C -1.6692,E1 24.8411,E2 262.6692} C_DIS
LIN {X -113.1114,Y -12.3335,Z 118,A -178.5829,B 24.9482,C -1.6619,E1 24.8405,E2 264.5961} C_DIS
LIN {X -113.4278,Y -8.9565,Z 118,A 179.6016,B 24.9482,C -1.6632,E1 24.8401,E2 266.4193} C_DIS
LIN {X -113.6673,Y -5.0842,Z 118,A 178.1176,B 24.9466,C -1.6878,E1 24.8399,E2 267.8536} C_DIS
LIN {X -113.7692,Y -1.6786,Z 118,A 176.533,B 24.9459,C -1.6985,E1 24.8398,E2 269.4222} C_DIS
LIN {X -113.7476,Y 2.8286,Z 118,A 173.7335,B 24.9468,C -1.6852,E1 24.8399,E2 272.2704} C_DIS
LIN {X -113.6181,Y 6.0863,Z 118,A 172.466,B 24.9455,C -1.7051,E1 24.8401,E2 273.4979} C_DIS
LIN {X -113.3653,Y 9.7377,Z 118,A 170.5959,B 24.9452,C -1.71,E1 24.8405,E2 275.3676} C_DIS
LIN {X -112.8284,Y 14.6915,Z 118,A 168.0992,B 24.9446,C -1.7187,E1 24.8413,E2 277.8585} C_DIS
LIN {X -112.3852,Y 17.7707,Z 118,A 166.3978,B 24.9446,C -1.7185,E1 24.842,E2 279.5706} C_DIS
LIN {X -111.6891,Y 21.718,Z 118,A 164.4894,B 24.944,C -1.7293,E1 24.843,E2 281.4645} C_DIS
LIN {X -110.9438,Y 25.2522,Z 118,A 162.6774,B 24.9436,C -1.7355,E1 24.844,E2 283.2726} C_DIS
LIN {X -110.1791,Y 28.4015,Z 118,A 161.0333,B 24.9432,C -1.7402,E1 24.8451,E2 284.9149} C_DIS
LIN {X -109.1728,Y 32.0543,Z 118,A 159.0601,B 24.943,C -1.7437,E1 24.8466,E2 286.8911} C_DIS
LIN {X -108.2432,Y 35.0639,Z 118,A 156.922,B 24.9441,C -1.7273,E1 24.8485,E2 289.0808} C_DIS
LIN {X -106.9006,Y 38.9659,Z 118,A 155.4035,B 24.9422,C -1.7555,E1 24.8499,E2 290.5406} C_DIS
LIN {X -105.5569,Y 42.4738,Z 118,A 153.6665,B 24.9415,C -1.7674,E1 24.8516,E2 292.2589} C_DIS
LIN {X -103.1405,Y 48.0428,Z 118,A 150.4184,B 24.9413,C -1.7692,E1 24.8553,E2 295.5206} C_DIS
LIN {X -101.4489,Y 51.5196,Z 118,A 148.522,B 24.9408,C -1.7771,E1 24.8576,E2 297.4085} C_DIS
LIN {X -99.1052,Y 55.897,Z 118,A 145.9595,B 24.9405,C -1.782,E1 24.8611,E2 299.9728} C_DIS
LIN {X -97.076,Y 59.35,Z 118,A 143.8176,B 24.9405,C -1.7829,E1 24.8641,E2 302.1237} C_DIS
LIN {X -95.027,Y 62.5776,Z 118,A 142.0849,B 24.9395,C -1.7959,E1 24.8667,E2 303.834} C_DIS
LIN {X -91.9406,Y 67.0302,Z 118,A 139.2557,B 24.9393,C -1.7995,E1 24.8713,E2 306.6686} C_DIS
LIN {X -88.3182,Y 71.7355,Z 118,A 136.2138,B 24.9389,C -1.8055,E1 24.8765,E2 309.7107} C_DIS
LIN {X -84.8255,Y 75.8334,Z 118,A 133.4563,B 24.9385,C -1.8106,E1 24.8815,E2 312.4683} C_DIS
LIN {X -80.671,Y 80.2397,Z 118,A 130.3639,B 24.9382,C -1.8165,E1 24.8875,E2 315.5602} C_DIS
LIN {X -78.1106,Y 82.7336,Z 118,A 128.7458,B 24.9374,C -1.8281,E1 24.8907,E2 317.1574} C_DIS
LIN {X -74.5386,Y 85.9665,Z 118,A 125.625,B 24.9389,C -1.806,E1 24.8974,E2 320.3431} C_DIS
LIN {X -71.4309,Y 88.5651,Z 118,A 124.149,B 24.937,C -1.833,E1 24.9005,E2 321.7605} C_DIS
LIN {X -68.0209,Y 91.2107,Z 118,A 121.8069,B 24.9372,C -1.8308,E1 24.9057,E2 324.1163} C_DIS
LIN {X -65.2149,Y 93.2374,Z 118,A 119.8699,B 24.9375,C -1.8266,E1 24.9102,E2 326.0699} C_DIS
LIN {X -60.8542,Y 96.142,Z 118,A 117.6178,B 24.936,C -1.8472,E1 24.9153,E2 328.2803} C_DIS
LIN {X -55.643,Y 99.247,Z 118,A 114.2011,B 24.9367,C -1.8381,E1 24.9236,E2 331.7288} C_DIS
LIN {X -51.6841,Y 101.3649,Z 118,A 112.1968,B 24.9357,C -1.8523,E1 24.9285,E2 333.705} C_DIS
LIN {X -49.5108,Y 102.4442,Z 118,A 110.4597,B 24.937,C -1.8334,E1 24.933,E2 335.4914} C_DIS
LIN {X -45.8969,Y 104.1142,Z 118,A 109.1401,B 24.9349,C -1.8642,E1 24.9362,E2 336.741} C_DIS
LIN {X -41.2416,Y 106.0441,Z 118,A 106.1213,B 24.936,C -1.8481,E1 24.9441,E2 339.8047} C_DIS
LIN {X -36.3196,Y 107.8284,Z 118,A 103.0165,B 24.9371,C -1.8324,E1 24.9525,E2 342.9528} C_DIS
LIN {X -31.4995,Y 109.3348,Z 118,A 101.1283,B 24.935,C -1.8619,E1 24.9573,E2 344.7741} C_DIS
LIN {X -27.9913,Y 110.2845,Z 118,A 99.3817,B 24.9346,C -1.8672,E1 24.962,E2 346.5107} C_DIS
LIN {X -25.0092,Y 111,Z 118,A 97.271,B 24.9362,C -1.8453,E1 24.9679,E2 348.6763} C_DIS
LIN {X -20.8965,Y 111.8472,Z 118,A 95.6398,B 24.9347,C -1.8669,E1 24.9723,E2 350.2579} C_DIS
LIN {X -17.9044,Y 112.3645,Z 118,A 93.4502,B 24.9365,C -1.8407,E1 24.9785,E2 352.5116} C_DIS
LIN {X -13.0571,Y 113.0293,Z 118,A 92.0601,B 24.9333,C -1.8867,E1 24.982,E2 353.7935} C_DIS
LIN {X -7.1736,Y 113.5556,Z 118,A 88.7768,B 24.9341,C -1.8751,E1 24.9912,E2 357.1058} C_DIS
LIN {X -0.5524,Y 113.7796,Z 118,A 85.8662,B 24.9327,C -1.894,E1 24.9992,E2 359.9719} C_DIS
LIN {X 5.546,Y 113.6475,Z 118,A 82.0476,B 24.935,C -1.8627,E1 25.0101,E2 363.8642} C_DIS
LIN {X 10.9761,Y 113.2514,Z 118,A 78.9157,B 24.9361,C -1.846,E1 25.0189,E2 367.0338} C_DIS
LIN {X 15.597,Y 112.7075,Z 118,A 77.2629,B 24.9341,C -1.8747,E1 25.0233,E2 368.6173} C_DIS
LIN {X 21.4452,Y 111.7416,Z 118,A 74.3286,B 24.9341,C -1.8758,E1 25.0314,E2 371.5459} C_DIS
LIN {X 25.7646,Y 110.8255,Z 118,A 72.0705,B 24.9342,C -1.8732,E1 25.0375,E2 373.8072} C_DIS
LIN {X 29.3992,Y 109.9174,Z 118,A 70.1883,B 24.9342,C -1.8722,E1 25.0426,E2 375.6889} C_DIS
LIN {X 32.3926,Y 109.0724,Z 118,A 68.6122,B 24.9344,C -1.8706,E1 25.0468,E2 377.2659} C_DIS
LIN {X 35.8243,Y 107.9954,Z 118,A 66.9277,B 24.9341,C -1.8746,E1 25.0513,E2 378.9378} C_DIS
LIN {X 39.4573,Y 106.7213,Z 118,A 64.9447,B 24.9344,C -1.871,E1 25.0565,E2 380.9255} C_DIS
LIN {X 42.7997,Y 105.4242,Z 118,A 63.0652,B 24.9347,C -1.8659,E1 25.0614,E2 382.8128} C_DIS
LIN {X 45.6529,Y 104.2206,Z 118,A 60.7794,B 24.937,C -1.8327,E1 25.0675,E2 385.1716} C_DIS
LIN {X 50.1026,Y 102.1569,Z 118,A 59.0483,B 24.935,C -1.8617,E1 25.0716,E2 386.8295} C_DIS
LIN {X 52.7561,Y 100.8115,Z 118,A 57.5396,B 24.9352,C -1.8593,E1 25.0754,E2 388.3398} C_DIS
LIN {X 58.5659,Y 97.5525,Z 118,A 54.1256,B 24.9357,C -1.8518,E1 25.0837,E2 391.7613} C_DIS
LIN {X 61.2642,Y 95.8792,Z 118,A 52.3378,B 24.9365,C -1.841,E1 25.0879,E2 393.5688} C_DIS
LIN {X 65.0544,Y 93.3489,Z 118,A 50.2795,B 24.936,C -1.8476,E1 25.0926,E2 395.6045} C_DIS
LIN {X 68.0944,Y 91.1555,Z 118,A 48.4319,B 24.9361,C -1.8461,E1 25.0968,E2 397.4493} C_DIS
LIN {X 70.656,Y 89.1842,Z 118,A 46.5873,B 24.937,C -1.8334,E1 25.1009,E2 399.3168} C_DIS
LIN {X 74.1629,Y 86.2912,Z 118,A 44.1428,B 24.9378,C -1.8221,E1 25.1061,E2 401.7787} C_DIS
LIN {X 76.6785,Y 84.0623,Z 118,A 42.3839,B 24.9382,C -1.8157,E1 25.1098,E2 403.5456} C_DIS
LIN {X 79.4959,Y 81.4058,Z 118,A 40.8221,B 24.9373,C -1.8288,E1 25.1128,E2 405.0699} C_DIS
LIN {X 81.4633,Y 79.4371,Z 118,A 39.1215,B 24.9384,C -1.8124,E1 25.1162,E2 406.802} C_DIS
LIN {X 83.7386,Y 77.0321,Z 118,A 37.7268,B 24.9379,C -1.8208,E1 25.1188,E2 408.1706} C_DIS
LIN {X 86.5159,Y 73.8992,Z 118,A 34.9371,B 24.9402,C -1.7855,E1 25.124,E2 411.0311} C_DIS
LIN {X 89.8871,Y 69.7606,Z 118,A 33.1097,B 24.9381,C -1.8175,E1 25.127,E2 412.7744} C_DIS
LIN {X 91.5833,Y 67.5183,Z 118,A 31.6548,B 24.9384,C -1.8122,E1 25.1294,E2 414.2348} C_DIS
LIN {X 93.2481,Y 65.1994,Z 118,A 29.9152,B 24.9396,C -1.7949,E1 25.1323,E2 416.0067} C_DIS
LIN {X 96.2843,Y 60.6266,Z 118,A 27.4109,B 24.9393,C -1.7994,E1 25.1361,E2 418.4878} C_DIS
LIN {X 98.3644,Y 57.1915,Z 118,A 25.4458,B 24.9395,C -1.7965,E1 25.1389,E2 420.4497} C_DIS
LIN {X 100.0232,Y 54.2349,Z 118,A 23.8185,B 24.9395,C -1.7955,E1 25.141,E2 422.0709} C_DIS
LIN {X 101.7305,Y 50.9628,Z 118,A 20.8005,B 24.9434,C -1.7379,E1 25.145,E2 425.2087} C_DIS
LIN {X 104.5795,Y 44.8295,Z 118,A 18.6277,B 24.9404,C -1.7837,E1 25.1473,E2 427.2614} C_DIS
LIN {X 106.8728,Y 39.0421,Z 118,A 15.392,B 24.9413,C -1.7699,E1 25.1506,E2 430.512} C_DIS
LIN {X 108.0555,Y 35.6442,Z 118,A 13.5849,B 24.9416,C -1.7646,E1 25.1522,E2 432.3213} C_DIS
LIN {X 108.9123,Y 32.9323,Z 118,A 12.1097,B 24.9421,C -1.7582,E1 25.1534,E2 433.803} C_DIS
LIN {X 109.949,Y 29.2823,Z 118,A 10.2558,B 24.9423,C -1.755,E1 25.1548,E2 435.6541} C_DIS
LIN {X 110.7507,Y 26.0884,Z 118,A 8.1329,B 24.944,C -1.7285,E1 25.1562,E2 437.827} C_DIS
LIN {X 111.6206,Y 22.0736,Z 118,A 6.3385,B 24.9436,C -1.7345,E1 25.1571,E2 439.5968} C_DIS
LIN {X 112.6816,Y 15.7793,Z 118,A 3.3522,B 24.9436,C -1.7348,E1 25.1584,E2 442.5649} C_DIS
LIN {X 113.4067,Y 9.2208,Z 118,A -0.3652,B 24.9455,C -1.706,E1 25.1595,E2 446.3282} C_DIS
LIN {X 113.6573,Y 5.3181,Z 118,A -1.9077,B 24.9446,C -1.7192,E1 25.1597,E2 447.8304} C_DIS
LIN {X 113.7614,Y 2.103,Z 118,A -3.9255,B 24.9461,C -1.6956,E1 25.1597,E2 449.8917} C_DIS
LIN {X 113.7674,Y -1.7743,Z 118,A -6.1438,B 24.9473,C -1.6771,E1 25.1597,E2 452.1405} C_DIS
LIN {X 113.5727,Y -6.9081,Z 118,A -7.9044,B 24.9454,C -1.7066,E1 25.1594,E2 453.821} C_DIS
LIN {X 112.8972,Y -14.1604,Z 118,A -11.413,B 24.9457,C -1.702,E1 25.1585,E2 457.3197} C_DIS
LIN {X 112.0714,Y -19.6544,Z 118,A -14.2004,B 24.9463,C -1.6933,E1 25.1573,E2 460.1112} C_DIS
LIN {X 111.3914,Y -23.1979,Z 118,A -16.8331,B 24.949,C -1.6499,E1 25.1558,E2 462.831} C_DIS
LIN {X 110.3466,Y -27.7498,Z 118,A -18.5371,B 24.9476,C -1.6721,E1 25.1547,E2 464.4729} C_DIS
LIN {X 109.5124,Y -30.8728,Z 118,A -19.9778,B 24.9474,C -1.6755,E1 25.1536,E2 465.8971} C_DIS
LIN {X 107.8428,Y -36.2768,Z 118,A -22.9608,B 24.9483,C -1.6602,E1 25.1511,E2 468.8992} C_DIS
LIN {X 106.6079,Y -39.7637,Z 118,A -24.874,B 24.9489,C -1.652,E1 25.1493,E2 470.821} C_DIS
LIN {X 105.4048,Y -42.8475,Z 118,A -27.0911,B 24.9507,C -1.6216,E1 25.1469,E2 473.0975} C_DIS
LIN {X 103.628,Y -46.9827,Z 118,A -28.6026,B 24.949,C -1.6493,E1 25.1453,E2 474.5355} C_DIS
LIN {X 101.6268,Y -51.1713,Z 118,A -31.1297,B 24.95,C -1.6335,E1 25.1421,E2 477.0865} C_DIS
LIN {X 99.9658,Y -54.3408,Z 118,A -33.3762,B 24.9516,C -1.6078,E1 25.1391,E2 479.3818} C_DIS
LIN {X 97.9258,Y -57.9363,Z 118,A -35.6377,B 24.9524,C -1.5935,E1 25.1358,E2 481.6653} C_DIS
LIN {X 95.2686,Y -62.2111,Z 118,A -37.5088,B 24.951,C -1.6165,E1 25.1331,E2 483.4727} C_DIS
LIN {X 92.8431,Y -65.7753,Z 118,A -40.0818,B 24.9525,C -1.5921,E1 25.1289,E2 486.0908} C_DIS
LIN {X 90.4733,Y -68.9999,Z 118,A -41.6464,B 24.9516,C -1.6071,E1 25.1264,E2 487.6124} C_DIS
LIN {X 88.2651,Y -71.801,Z 118,A -43.3407,B 24.9516,C -1.607,E1 25.1234,E2 489.2992} C_DIS
LIN {X 86.1312,Y -74.35,Z 118,A -45.0546,B 24.952,C -1.6007,E1 25.1203,E2 491.0201} C_DIS
LIN {X 83.8976,Y -76.8588,Z 118,A -46.6973,B 24.9521,C -1.5986,E1 25.1172,E2 492.6603} C_DIS
LIN {X 81.4657,Y -79.4345,Z 118,A -48.4102,B 24.9521,C -1.5974,E1 25.1139,E2 494.3689} C_DIS
LIN {X 79.0371,Y -81.8488,Z 118,A -50.1792,B 24.9526,C -1.5912,E1 25.1104,E2 496.1452} C_DIS
LIN {X 76.4451,Y -84.2772,Z 118,A -52.0876,B 24.9531,C -1.5814,E1 25.1064,E2 498.0688} C_DIS
LIN {X 73.8021,Y -86.5987,Z 118,A -53.7228,B 24.9531,C -1.5836,E1 25.103,E2 499.6925} C_DIS
LIN {X 70.924,Y -88.9724,Z 118,A -55.631,B 24.9533,C -1.578,E1 25.0989,E2 501.6065} C_DIS
LIN {X 68.2475,Y -91.0405,Z 118,A -57.2917,B 24.9534,C -1.5763,E1 25.0952,E2 503.2654} C_DIS
LIN {X 65.9565,Y -92.7137,Z 118,A -59.6165,B 24.956,C -1.5331,E1 25.0897,E2 505.684} C_DIS
LIN {X 61.2972,Y -95.858,Z 118,A -61.525,B 24.9539,C -1.5688,E1 25.0854,E2 507.5021} C_DIS
LIN {X 58.218,Y -97.7593,Z 118,A -63.396,B 24.9542,C -1.5631,E1 25.0809,E2 509.3805} C_DIS
LIN {X 55.3791,Y -99.3944,Z 118,A -64.8158,B 24.9538,C -1.5705,E1 25.0775,E2 510.7787} C_DIS
LIN {X 53.2365,Y -100.5585,Z 118,A -66.1591,B 24.9542,C -1.5632,E1 25.0742,E2 512.1354} C_DIS
LIN {X 50.3514,Y -102.0336,Z 118,A -67.8938,B 24.9546,C -1.5558,E1 25.0698,E2 513.8828} C_DIS
LIN {X 45.2817,Y -104.3824,Z 118,A -71.0928,B 24.9559,C -1.5343,E1 25.0616,E2 517.1246} C_DIS
LIN {X 41.9185,Y -105.7782,Z 118,A -72.252,B 24.9543,C -1.5617,E1 25.0588,E2 518.2166} C_DIS
LIN {X 37.3436,Y -107.4786,Z 118,A -75.0366,B 24.9553,C -1.5438,E1 25.0514,E2 521.0376} C_DIS
LIN {X 33.8557,Y -108.6273,Z 118,A -76.8508,B 24.9553,C -1.5431,E1 25.0465,E2 522.8501} C_DIS
LIN {X 30.1304,Y -109.7199,Z 118,A -78.8085,B 24.9555,C -1.5408,E1 25.0413,E2 524.8099} C_DIS
LIN {X 26.6061,Y -110.627,Z 118,A -80.3652,B 24.9549,C -1.5512,E1 25.0371,E2 526.3399} C_DIS
LIN {X 20.8455,Y -111.8571,Z 118,A -84.2447,B 24.9574,C -1.5086,E1 25.0262,E2 530.3154} C_DIS
LIN {X 16.1191,Y -112.6333,Z 118,A -85.5917,B 24.9548,C -1.5533,E1 25.0228,E2 531.5552} C_DIS
LIN {X 8.9547,Y -113.428,Z 118,A -89.1131,B 24.9546,C -1.5558,E1 25.0131,E2 535.0682} C_DIS
LIN {X 2.7365,Y -113.7497,Z 118,A -92.5904,B 24.9556,C -1.5396,E1 25.0033,E2 538.5828} C_DIS
LIN {X 0.8048,Y -113.7717,Z 118,A -93.5748,B 24.9556,C -1.539,E1 25.0005,E2 539.5686} C_DIS
Enddeposition()
END
